    LOCAL CONST Robtarget Tr_meulage_motif_1_369 := [[-197.1254375,6.42979248046875,2.70970288085938],[0.587839766788017,-0.597604018313253,0.388723125784971,-0.382371778977509],[0,0,0,0],[8.999999E+09,8.999999E+09,8.999999E+09,8.999999E+09,8.999999E+09,8.999999E+09]];
    LOCAL CONST Robtarget Tr_meulage_motif_1_370 := [[-197.496625,7.3583505859375,2.7097021484375],[0.587839766788017,-0.597604018313253,0.388723125784971,-0.382371778977509],[0,0,0,0],[8.999999E+09,8.999999E+09,8.999999E+09,8.999999E+09,8.999999E+09,8.999999E+09]];
    LOCAL CONST Robtarget Tr_meulage_motif_1_371 := [[-197.8661875,8.279548828125,2.5990986328125],[0.587839766788017,-0.597604018313253,0.388723125784971,-0.382371778977509],[0,0,0,0],[8.999999E+09,8.999999E+09,8.999999E+09,8.999999E+09,8.999999E+09,8.999999E+09]];
    LOCAL CONST Robtarget Tr_meulage_motif_1_372 := [[-198.2196875,9.1575625,2.38792309570313],[0.587839766788017,-0.597604018313253,0.388723125784971,-0.382371778977509],[0,0,0,0],[8.999999E+09,8.999999E+09,8.999999E+09,8.999999E+09,8.999999E+09,8.999999E+09]];
    LOCAL CONST Robtarget Tr_meulage_motif_1_373 := [[-198.538984375,9.9482470703125,2.11611083984375],[0.587839766788017,-0.597604018313253,0.388723125784971,-0.382371778977509],[0,0,0,0],[8.999999E+09,8.999999E+09,8.999999E+09,8.999999E+09,8.999999E+09,8.999999E+09]];
    LOCAL CONST Robtarget Tr_meulage_motif_1_374 := [[-198.806203125,10.6076689453125,1.81198828125],[0.587839766788017,-0.597604018313253,0.388723125784971,-0.382371778977509],[0,0,0,0],[8.999999E+09,8.999999E+09,8.999999E+09,8.999999E+09,8.999999E+09,8.999999E+09]];
    LOCAL CONST Robtarget Tr_meulage_motif_1_375 := [[-199.196984375,11.5655166015625,1.14949658203125],[0.587839766788017,-0.597604018313253,0.388723125784971,-0.382371778977509],[0,0,0,0],[8.999999E+09,8.999999E+09,8.999999E+09,8.999999E+09,8.999999E+09,8.999999E+09]];
    LOCAL CONST Robtarget Tr_meulage_motif_1_376 := [[-199.541015625,12.3993203125,0.247597717285156],[0.587839766788017,-0.597604018313253,0.388723125784971,-0.382371778977509],[0,0,0,0],[8.999999E+09,8.999999E+09,8.999999E+09,8.999999E+09,8.999999E+09,8.999999E+09]];
    LOCAL CONST Robtarget Tr_meulage_motif_1_377 := [[-199.7503125,12.89178125,-0.798370178222656],[0.587839766788017,-0.597604018313253,0.388723125784971,-0.382371778977509],[0,0,0,0],[8.999999E+09,8.999999E+09,8.999999E+09,8.999999E+09,8.999999E+09,8.999999E+09]];
    LOCAL CONST Robtarget Tr_meulage_motif_1_378 := [[-199.792984375,12.9777431640625,-1.49615588378906],[0.587839766788017,-0.597604018313253,0.388723125784971,-0.382371778977509],[0,0,0,0],[8.999999E+09,8.999999E+09,8.999999E+09,8.999999E+09,8.999999E+09,8.999999E+09]];
    LOCAL CONST Robtarget Tr_meulage_motif_1_379 := [[-199.76965625,12.9004716796875,-2.13255444335937],[0.587839766788017,-0.597604018313253,0.388723125784971,-0.382371778977509],[0,0,0,0],[8.999999E+09,8.999999E+09,8.999999E+09,8.999999E+09,8.999999E+09,8.999999E+09]];
    LOCAL CONST Robtarget Tr_meulage_motif_1_380 := [[-199.738171875,12.8063076171875,-2.64972607421875],[0.587839766788017,-0.597604018313253,0.388723125784971,-0.382371778977509],[0,0,0,0],[8.999999E+09,8.999999E+09,8.999999E+09,8.999999E+09,8.999999E+09,8.999999E+09]];
    LOCAL CONST Robtarget Tr_meulage_motif_1_381 := [[-199.526421875,12.2498720703125,-3.54807690429688],[0.587839766788017,-0.597604018313253,0.388723125784971,-0.382371778977509],[0,0,0,0],[8.999999E+09,8.999999E+09,8.999999E+09,8.999999E+09,8.999999E+09,8.999999E+09]];
    LOCAL CONST Robtarget Tr_meulage_motif_1_382 := [[-199.35234375,11.8015830078125,-3.97934716796875],[0.587839766788017,-0.597604018313253,0.388723125784971,-0.382371778977509],[0,0,0,0],[8.999999E+09,8.999999E+09,8.999999E+09,8.999999E+09,8.999999E+09,8.999999E+09]];
    LOCAL CONST Robtarget Tr_meulage_motif_1_383 := [[-198.956453125,10.7936171875,-4.57071630859375],[0.587839766788017,-0.597604018313253,0.388723125784971,-0.382371778977509],[0,0,0,0],[8.999999E+09,8.999999E+09,8.999999E+09,8.999999E+09,8.999999E+09,8.999999E+09]];
    LOCAL CONST Robtarget Tr_meulage_motif_1_384 := [[-198.65303125,10.025794921875,-4.86619775390625],[0.587839766788017,-0.597604018313253,0.388723125784971,-0.382371778977509],[0,0,0,0],[8.999999E+09,8.999999E+09,8.999999E+09,8.999999E+09,8.999999E+09,8.999999E+09]];
    LOCAL CONST Robtarget Tr_meulage_motif_1_385 := [[-198.309171875,9.1595400390625,-5.0706689453125],[0.587839766788017,-0.597604018313253,0.388723125784971,-0.382371778977509],[0,0,0,0],[8.999999E+09,8.999999E+09,8.999999E+09,8.999999E+09,8.999999E+09,8.999999E+09]];
    LOCAL CONST Robtarget Tr_meulage_motif_1_386 := [[-197.945953125,8.247658203125,-5.17920849609375],[0.587839766788017,-0.597604018313253,0.388723125784971,-0.382371778977509],[0,0,0,0],[8.999999E+09,8.999999E+09,8.999999E+09,8.999999E+09,8.999999E+09,8.999999E+09]];
    LOCAL CONST Robtarget Tr_meulage_motif_1_387 := [[-197.57865625,7.325552734375,-5.28981005859375],[0.587839766788017,-0.597604018313253,0.388723125784971,-0.382371778977509],[0,0,0,0],[8.999999E+09,8.999999E+09,8.999999E+09,8.999999E+09,8.999999E+09,8.999999E+09]];
    LOCAL CONST Robtarget Tr_meulage_motif_1_388 := [[-197.20746875,6.3969951171875,-5.28980908203125],[0.587839766788017,-0.597604018313253,0.388723125784971,-0.382371778977509],[0,0,0,0],[8.999999E+09,8.999999E+09,8.999999E+09,8.999999E+09,8.999999E+09,8.999999E+09]];
    LOCAL CONST Robtarget Tr_meulage_motif_1_389 := [[-196.83628125,5.46843701171875,-5.28980859375],[0.587839766788017,-0.597604018313253,0.388723125784971,-0.382371778977509],[0,0,0,0],[8.999999E+09,8.999999E+09,8.999999E+09,8.999999E+09,8.999999E+09,8.999999E+09]];
    LOCAL CONST Robtarget Tr_meulage_motif_1_390 := [[-196.46509375,4.53987939453125,-5.2898076171875],[0.587839766788017,-0.597604018313253,0.388723125784971,-0.382371778977509],[0,0,0,0],[8.999999E+09,8.999999E+09,8.999999E+09,8.999999E+09,8.999999E+09,8.999999E+09]];
    LOCAL CONST Robtarget Tr_meulage_motif_1_391 := [[-196.09390625,3.61132153320312,-5.289806640625],[0.587839766788017,-0.597604018313253,0.388723125784971,-0.382371778977509],[0,0,0,0],[8.999999E+09,8.999999E+09,8.999999E+09,8.999999E+09,8.999999E+09,8.999999E+09]];
    LOCAL CONST Robtarget Tr_meulage_motif_1_392 := [[-195.72271875,2.682763671875,-5.28980615234375],[0.587839766788017,-0.597604018313253,0.388723125784971,-0.382371778977509],[0,0,0,0],[8.999999E+09,8.999999E+09,8.999999E+09,8.999999E+09,8.999999E+09,8.999999E+09]];
    LOCAL CONST Robtarget Tr_meulage_motif_1_393 := [[-195.35153125,1.75420581054687,-5.28980517578125],[0.587839766788017,-0.597604018313253,0.388723125784971,-0.382371778977509],[0,0,0,0],[8.999999E+09,8.999999E+09,8.999999E+09,8.999999E+09,8.999999E+09,8.999999E+09]];
    LOCAL CONST Robtarget Tr_meulage_motif_1_394 := [[-194.98034375,0.825648010253906,-5.28980419921875],[0.587839766788017,-0.597604018313253,0.388723125784971,-0.382371778977509],[0,0,0,0],[8.999999E+09,8.999999E+09,8.999999E+09,8.999999E+09,8.999999E+09,8.999999E+09]];
    LOCAL CONST Robtarget Tr_meulage_motif_1_395 := [[-194.60915625,-0.102909828186035,-5.2898037109375],[0.587839766788017,-0.597604018313253,0.388723125784971,-0.382371778977509],[0,0,0,0],[8.999999E+09,8.999999E+09,8.999999E+09,8.999999E+09,8.999999E+09,8.999999E+09]];
    LOCAL CONST Robtarget Tr_meulage_motif_1_396 := [[-194.23796875,-1.03146765136719,-5.289802734375],[0.587839766788017,-0.597604018313253,0.388723125784971,-0.382371778977509],[0,0,0,0],[8.999999E+09,8.999999E+09,8.999999E+09,8.999999E+09,8.999999E+09,8.999999E+09]];
    LOCAL CONST Robtarget Tr_meulage_motif_1_397 := [[-193.86678125,-1.96002551269531,-5.2898017578125],[0.587839766788017,-0.597604018313253,0.388723125784971,-0.382371778977509],[0,0,0,0],[8.999999E+09,8.999999E+09,8.999999E+09,8.999999E+09,8.999999E+09,8.999999E+09]];
    LOCAL CONST Robtarget Tr_meulage_motif_1_398 := [[-193.49559375,-2.88858325195313,-5.28980126953125],[0.587839766788017,-0.597604018313253,0.388723125784971,-0.382371778977509],[0,0,0,0],[8.999999E+09,8.999999E+09,8.999999E+09,8.999999E+09,8.999999E+09,8.999999E+09]];
    LOCAL CONST Robtarget Tr_meulage_motif_1_399 := [[-193.12440625,-3.81714111328125,-5.28980029296875],[0.587839766788017,-0.597604018313253,0.388723125784971,-0.382371778977509],[0,0,0,0],[8.999999E+09,8.999999E+09,8.999999E+09,8.999999E+09,8.999999E+09,8.999999E+09]];
    LOCAL CONST Robtarget Tr_meulage_motif_1_400 := [[-192.75321875,-4.74569873046875,-5.28979931640625],[0.587839766788017,-0.597604018313253,0.388723125784971,-0.382371778977509],[0,0,0,0],[8.999999E+09,8.999999E+09,8.999999E+09,8.999999E+09,8.999999E+09,8.999999E+09]];
    LOCAL CONST Robtarget Tr_meulage_motif_1_401 := [[-192.38203125,-5.6742568359375,-5.289798828125],[0.587839766788017,-0.597604018313253,0.388723125784971,-0.382371778977509],[0,0,0,0],[8.999999E+09,8.999999E+09,8.999999E+09,8.999999E+09,8.999999E+09,8.999999E+09]];
    LOCAL CONST Robtarget Tr_meulage_motif_1_402 := [[-192.01084375,-6.602814453125,-5.2897978515625],[0.587839766788017,-0.597604018313253,0.388723125784971,-0.382371778977509],[0,0,0,0],[8.999999E+09,8.999999E+09,8.999999E+09,8.999999E+09,8.999999E+09,8.999999E+09]];
    LOCAL CONST Robtarget Tr_meulage_motif_1_403 := [[-191.63965625,-7.53137255859375,-5.289796875],[0.587839766788017,-0.597604018313253,0.388723125784971,-0.382371778977509],[0,0,0,0],[8.999999E+09,8.999999E+09,8.999999E+09,8.999999E+09,8.999999E+09,8.999999E+09]];
    LOCAL CONST Robtarget Tr_meulage_motif_1_404 := [[-191.268453125,-8.4599306640625,-5.28979638671875],[0.587839766788017,-0.597604018313253,0.388723125784971,-0.382371778977509],[0,0,0,0],[8.999999E+09,8.999999E+09,8.999999E+09,8.999999E+09,8.999999E+09,8.999999E+09]];
    LOCAL CONST Robtarget Tr_meulage_motif_1_405 := [[-190.897265625,-9.38848828125,-5.28979541015625],[0.587839766788017,-0.597604018313253,0.388723125784971,-0.382371778977509],[0,0,0,0],[8.999999E+09,8.999999E+09,8.999999E+09,8.999999E+09,8.999999E+09,8.999999E+09]];
    LOCAL CONST Robtarget Tr_meulage_motif_1_406 := [[-190.526078125,-10.3170458984375,-5.28979443359375],[0.587839766788017,-0.597604018313253,0.388723125784971,-0.382371778977509],[0,0,0,0],[8.999999E+09,8.999999E+09,8.999999E+09,8.999999E+09,8.999999E+09,8.999999E+09]];
    LOCAL CONST Robtarget Tr_meulage_motif_1_407 := [[-190.154890625,-11.245603515625,-5.28979345703125],[0.587839766788017,-0.597604018313253,0.388723125784971,-0.382371778977509],[0,0,0,0],[8.999999E+09,8.999999E+09,8.999999E+09,8.999999E+09,8.999999E+09,8.999999E+09]];
    LOCAL CONST Robtarget Tr_meulage_motif_1_408 := [[-189.783703125,-12.1741611328125,-5.28979296875],[0.587839766788017,-0.597604018313253,0.388723125784971,-0.382371778977509],[0,0,0,0],[8.999999E+09,8.999999E+09,8.999999E+09,8.999999E+09,8.999999E+09,8.999999E+09]];
    LOCAL CONST Robtarget Tr_meulage_motif_1_409 := [[-189.412515625,-13.1027197265625,-5.2897919921875],[0.587839766788017,-0.597604018313253,0.388723125784971,-0.382371778977509],[0,0,0,0],[8.999999E+09,8.999999E+09,8.999999E+09,8.999999E+09,8.999999E+09,8.999999E+09]];
    LOCAL CONST Robtarget Tr_meulage_motif_1_410 := [[-189.041328125,-14.03127734375,-5.289791015625],[0.587839766788017,-0.597604018313253,0.388723125784971,-0.382371778977509],[0,0,0,0],[8.999999E+09,8.999999E+09,8.999999E+09,8.999999E+09,8.999999E+09,8.999999E+09]];
    LOCAL CONST Robtarget Tr_meulage_motif_1_411 := [[-188.670140625,-14.9598349609375,-5.28979052734375],[0.587839766788017,-0.597604018313253,0.388723125784971,-0.382371778977509],[0,0,0,0],[8.999999E+09,8.999999E+09,8.999999E+09,8.999999E+09,8.999999E+09,8.999999E+09]];
    LOCAL CONST Robtarget Tr_meulage_motif_1_412 := [[-188.298953125,-15.888392578125,-5.28978955078125],[0.587839766788017,-0.597604018313253,0.388723125784971,-0.382371778977509],[0,0,0,0],[8.999999E+09,8.999999E+09,8.999999E+09,8.999999E+09,8.999999E+09,8.999999E+09]];
    LOCAL CONST Robtarget Tr_meulage_motif_1_413 := [[-187.927765625,-16.816951171875,-5.28978857421875],[0.587839766788017,-0.597604018313253,0.388723125784971,-0.382371778977509],[0,0,0,0],[8.999999E+09,8.999999E+09,8.999999E+09,8.999999E+09,8.999999E+09,8.999999E+09]];
    LOCAL CONST Robtarget Tr_meulage_motif_1_414 := [[-187.556578125,-17.7455078125,-5.2897880859375],[0.587839766788017,-0.597604018313253,0.388723125784971,-0.382371778977509],[0,0,0,0],[8.999999E+09,8.999999E+09,8.999999E+09,8.999999E+09,8.999999E+09,8.999999E+09]];
    LOCAL CONST Robtarget Tr_meulage_motif_1_415 := [[-187.185390625,-18.67406640625,-5.289787109375],[0.587839766788017,-0.597604018313253,0.388723125784971,-0.382371778977509],[0,0,0,0],[8.999999E+09,8.999999E+09,8.999999E+09,8.999999E+09,8.999999E+09,8.999999E+09]];
    LOCAL CONST Robtarget Tr_meulage_motif_1_416 := [[-186.814203125,-19.602625,-5.2897861328125],[0.587839766788017,-0.597604018313253,0.388723125784971,-0.382371778977509],[0,0,0,0],[8.999999E+09,8.999999E+09,8.999999E+09,8.999999E+09,8.999999E+09,8.999999E+09]];
    LOCAL CONST Robtarget Tr_meulage_motif_1_417 := [[-186.443015625,-20.531181640625,-5.28978564453125],[0.587839766788017,-0.597604018313253,0.388723125784971,-0.382371778977509],[0,0,0,0],[8.999999E+09,8.999999E+09,8.999999E+09,8.999999E+09,8.999999E+09,8.999999E+09]];
    LOCAL CONST Robtarget Tr_meulage_motif_1_418 := [[-186.071828125,-21.459740234375,-5.28978466796875],[0.587839766788017,-0.597604018313253,0.388723125784971,-0.382371778977509],[0,0,0,0],[8.999999E+09,8.999999E+09,8.999999E+09,8.999999E+09,8.999999E+09,8.999999E+09]];
    LOCAL CONST Robtarget Tr_meulage_motif_1_419 := [[-185.700640625,-22.388296875,-5.28978369140625],[0.587839766788017,-0.597604018313253,0.388723125784971,-0.382371778977509],[0,0,0,0],[8.999999E+09,8.999999E+09,8.999999E+09,8.999999E+09,8.999999E+09,8.999999E+09]];
    LOCAL CONST Robtarget Tr_meulage_motif_1_420 := [[-185.329453125,-23.31685546875,-5.289783203125],[0.587839766788017,-0.597604018313253,0.388723125784971,-0.382371778977509],[0,0,0,0],[8.999999E+09,8.999999E+09,8.999999E+09,8.999999E+09,8.999999E+09,8.999999E+09]];
    LOCAL CONST Robtarget Tr_meulage_motif_1_421 := [[-184.958265625,-24.2454140625,-5.2897822265625],[0.587839766788017,-0.597604018313253,0.388723125784971,-0.382371778977509],[0,0,0,0],[8.999999E+09,8.999999E+09,8.999999E+09,8.999999E+09,8.999999E+09,8.999999E+09]];
    LOCAL CONST Robtarget Tr_meulage_motif_1_422 := [[-184.587078125,-25.173970703125,-5.28978125],[0.587839766788017,-0.597604018313253,0.388723125784971,-0.382371778977509],[0,0,0,0],[8.999999E+09,8.999999E+09,8.999999E+09,8.999999E+09,8.999999E+09,8.999999E+09]];
    LOCAL CONST Robtarget Tr_meulage_motif_1_423 := [[-184.215890625,-26.102529296875,-5.28978076171875],[0.587839766788017,-0.597604018313253,0.388723125784971,-0.382371778977509],[0,0,0,0],[8.999999E+09,8.999999E+09,8.999999E+09,8.999999E+09,8.999999E+09,8.999999E+09]];
    LOCAL CONST Robtarget Tr_meulage_motif_1_424 := [[-183.844703125,-27.0310859375,-5.28977978515625],[0.587839766788017,-0.597604018313253,0.388723125784971,-0.382371778977509],[0,0,0,0],[8.999999E+09,8.999999E+09,8.999999E+09,8.999999E+09,8.999999E+09,8.999999E+09]];
    LOCAL CONST Robtarget Tr_meulage_motif_1_425 := [[-183.473515625,-27.95964453125,-5.28977880859375],[0.587839766788017,-0.597604018313253,0.388723125784971,-0.382371778977509],[0,0,0,0],[8.999999E+09,8.999999E+09,8.999999E+09,8.999999E+09,8.999999E+09,8.999999E+09]];
    LOCAL CONST Robtarget Tr_meulage_motif_1_426 := [[-183.102328125,-28.888203125,-5.28977783203125],[0.587839766788017,-0.597604018313253,0.388723125784971,-0.382371778977509],[0,0,0,0],[8.999999E+09,8.999999E+09,8.999999E+09,8.999999E+09,8.999999E+09,8.999999E+09]];
    LOCAL CONST Robtarget Tr_meulage_motif_1_427 := [[-182.731140625,-29.816759765625,-5.28977734375],[0.587839766788017,-0.597604018313253,0.388723125784971,-0.382371778977509],[0,0,0,0],[8.999999E+09,8.999999E+09,8.999999E+09,8.999999E+09,8.999999E+09,8.999999E+09]];
    LOCAL CONST Robtarget Tr_meulage_motif_1_428 := [[-182.359953125,-30.745318359375,-5.2897763671875],[0.587839766788017,-0.597604018313253,0.388723125784971,-0.382371778977509],[0,0,0,0],[8.999999E+09,8.999999E+09,8.999999E+09,8.999999E+09,8.999999E+09,8.999999E+09]];
    LOCAL CONST Robtarget Tr_meulage_motif_1_429 := [[-181.988765625,-31.673875,-5.289775390625],[0.587839766788017,-0.597604018313253,0.388723125784971,-0.382371778977509],[0,0,0,0],[8.999999E+09,8.999999E+09,8.999999E+09,8.999999E+09,8.999999E+09,8.999999E+09]];
    LOCAL CONST Robtarget Tr_meulage_motif_1_430 := [[-181.617578125,-32.60243359375,-5.28977490234375],[0.587839766788017,-0.597604018313253,0.388723125784971,-0.382371778977509],[0,0,0,0],[8.999999E+09,8.999999E+09,8.999999E+09,8.999999E+09,8.999999E+09,8.999999E+09]];
    LOCAL CONST Robtarget Tr_meulage_motif_1_431 := [[-181.246390625,-33.5309921875,-5.28977392578125],[0.587839766788017,-0.597604018313253,0.388723125784971,-0.382371778977509],[0,0,0,0],[8.999999E+09,8.999999E+09,8.999999E+09,8.999999E+09,8.999999E+09,8.999999E+09]];
    LOCAL CONST Robtarget Tr_meulage_motif_1_432 := [[-180.875203125,-34.45955078125,-5.28977294921875],[0.587839766788017,-0.597604018313253,0.388723125784971,-0.382371778977509],[0,0,0,0],[8.999999E+09,8.999999E+09,8.999999E+09,8.999999E+09,8.999999E+09,8.999999E+09]];
    LOCAL CONST Robtarget Tr_meulage_motif_1_433 := [[-180.504015625,-35.38810546875,-5.2897724609375],[0.587839766788017,-0.597604018313253,0.388723125784971,-0.382371778977509],[0,0,0,0],[8.999999E+09,8.999999E+09,8.999999E+09,8.999999E+09,8.999999E+09,8.999999E+09]];
    LOCAL CONST Robtarget Tr_meulage_motif_1_434 := [[-180.132828125,-36.3166640625,-5.289771484375],[0.587839766788017,-0.597604018313253,0.388723125784971,-0.382371778977509],[0,0,0,0],[8.999999E+09,8.999999E+09,8.999999E+09,8.999999E+09,8.999999E+09,8.999999E+09]];
    LOCAL CONST Robtarget Tr_meulage_motif_1_435 := [[-179.761640625,-37.24522265625,-5.2897705078125],[0.587839766788017,-0.597604018313253,0.388723125784971,-0.382371778977509],[0,0,0,0],[8.999999E+09,8.999999E+09,8.999999E+09,8.999999E+09,8.999999E+09,8.999999E+09]];
    LOCAL CONST Robtarget Tr_meulage_motif_1_436 := [[-179.390453125,-38.17378125,-5.28977001953125],[0.587839766788017,-0.597604018313253,0.388723125784971,-0.382371778977509],[0,0,0,0],[8.999999E+09,8.999999E+09,8.999999E+09,8.999999E+09,8.999999E+09,8.999999E+09]];
    LOCAL CONST Robtarget Tr_meulage_motif_1_437 := [[-179.02315625,-39.09588671875,-5.40037158203125],[0.587839766788017,-0.597604018313253,0.388723125784971,-0.382371778977509],[0,0,0,0],[8.999999E+09,8.999999E+09,8.999999E+09,8.999999E+09,8.999999E+09,8.999999E+09]];
    LOCAL CONST Robtarget Tr_meulage_motif_1_438 := [[-178.659921875,-40.00776953125,-5.5089111328125],[0.587839766788017,-0.597604018313253,0.388723125784971,-0.382371778977509],[0,0,0,0],[8.999999E+09,8.999999E+09,8.999999E+09,8.999999E+09,8.999999E+09,8.999999E+09]];
    LOCAL CONST Robtarget Tr_meulage_motif_1_439 := [[-178.297125,-40.9182109375,-5.605623046875],[0.587839766788017,-0.597604018313253,0.388723125784971,-0.382371778977509],[0,0,0,0],[8.999999E+09,8.999999E+09,8.999999E+09,8.999999E+09,8.999999E+09,8.999999E+09]];
    LOCAL CONST Robtarget Tr_meulage_motif_1_440 := [[-177.940921875,-41.81337890625,-5.74241064453125],[0.587839766788017,-0.597604018313253,0.388723125784971,-0.382371778977509],[0,0,0,0],[8.999999E+09,8.999999E+09,8.999999E+09,8.999999E+09,8.999999E+09,8.999999E+09]];
    LOCAL CONST Robtarget Tr_meulage_motif_1_441 := [[-177.515703125,-42.88446875,-5.99027001953125],[0.587839766788017,-0.597604018313253,0.388723125784971,-0.382371778977509],[0,0,0,0],[8.999999E+09,8.999999E+09,8.999999E+09,8.999999E+09,8.999999E+09,8.999999E+09]];
    LOCAL CONST Robtarget Tr_meulage_motif_1_442 := [[-177.1755,-43.74487890625,-6.305171875],[0.587839766788017,-0.597604018313253,0.388723125784971,-0.382371778977509],[0,0,0,0],[8.999999E+09,8.999999E+09,8.999999E+09,8.999999E+09,8.999999E+09,8.999999E+09]];

    !Tr_meulage_motif_2 : Meulage d'un motif
    LOCAL CONST Robtarget Tr_meulage_motif_2_0 := [[111.493109375,113.3949609375,1.99855541992188],[-0.000489514218315733,0.0476030487198184,-0.010271051450657,-0.998813403809994],[0,0,0,0],[8.999999E+09,8.999999E+09,8.999999E+09,8.999999E+09,8.999999E+09,8.999999E+09]];
    LOCAL CONST Robtarget Tr_meulage_motif_2_1 := [[110.787296875,112.68659375,1.99164038085938],[-0.000489514218315733,0.0476030487198184,-0.010271051450657,-0.998813403809994],[0,0,0,0],[8.999999E+09,8.999999E+09,8.999999E+09,8.999999E+09,8.999999E+09,8.999999E+09]];
    LOCAL CONST Robtarget Tr_meulage_motif_2_2 := [[110.081484375,111.978234375,1.98472546386719],[-0.000489514218315733,0.0476030487198184,-0.010271051450657,-0.998813403809994],[0,0,0,0],[8.999999E+09,8.999999E+09,8.999999E+09,8.999999E+09,8.999999E+09,8.999999E+09]];
    LOCAL CONST Robtarget Tr_meulage_motif_2_3 := [[109.3756640625,111.2698671875,1.977810546875],[-0.000489514218315733,0.0476030487198184,-0.010271051450657,-0.998813403809994],[0,0,0,0],[8.999999E+09,8.999999E+09,8.999999E+09,8.999999E+09,8.999999E+09,8.999999E+09]];
    LOCAL CONST Robtarget Tr_meulage_motif_2_4 := [[108.6698515625,110.5615078125,1.9708955078125],[-0.000489514218315733,0.0476030487198184,-0.010271051450657,-0.998813403809994],[0,0,0,0],[8.999999E+09,8.999999E+09,8.999999E+09,8.999999E+09,8.999999E+09,8.999999E+09]];
    LOCAL CONST Robtarget Tr_meulage_motif_2_5 := [[107.9640390625,109.8531484375,1.96398059082031],[-0.000489514218315733,0.0476030487198184,-0.010271051450657,-0.998813403809994],[0,0,0,0],[8.999999E+09,8.999999E+09,8.999999E+09,8.999999E+09,8.999999E+09,8.999999E+09]];
    LOCAL CONST Robtarget Tr_meulage_motif_2_6 := [[107.25821875,109.14478125,1.95706567382813],[-0.000489514218315733,0.0476030487198184,-0.010271051450657,-0.998813403809994],[0,0,0,0],[8.999999E+09,8.999999E+09,8.999999E+09,8.999999E+09,8.999999E+09,8.999999E+09]];
    LOCAL CONST Robtarget Tr_meulage_motif_2_7 := [[106.55240625,108.436421875,1.95015075683594],[-0.000489514218315733,0.0476030487198184,-0.010271051450657,-0.998813403809994],[0,0,0,0],[8.999999E+09,8.999999E+09,8.999999E+09,8.999999E+09,8.999999E+09,8.999999E+09]];
    LOCAL CONST Robtarget Tr_meulage_motif_2_8 := [[105.84659375,107.7280546875,1.94323571777344],[-0.000489514218315733,0.0476030487198184,-0.010271051450657,-0.998813403809994],[0,0,0,0],[8.999999E+09,8.999999E+09,8.999999E+09,8.999999E+09,8.999999E+09,8.999999E+09]];
    LOCAL CONST Robtarget Tr_meulage_motif_2_9 := [[105.1407734375,107.0196953125,1.93632080078125],[-0.000489514218315733,0.0476030487198184,-0.010271051450657,-0.998813403809994],[0,0,0,0],[8.999999E+09,8.999999E+09,8.999999E+09,8.999999E+09,8.999999E+09,8.999999E+09]];
    LOCAL CONST Robtarget Tr_meulage_motif_2_10 := [[104.4349609375,106.3113359375,1.92940588378906],[-0.000489514218315733,0.0476030487198184,-0.010271051450657,-0.998813403809994],[0,0,0,0],[8.999999E+09,8.999999E+09,8.999999E+09,8.999999E+09,8.999999E+09,8.999999E+09]];
    LOCAL CONST Robtarget Tr_meulage_motif_2_11 := [[103.7291484375,105.60296875,1.92249084472656],[-0.000489514218315733,0.0476030487198184,-0.010271051450657,-0.998813403809994],[0,0,0,0],[8.999999E+09,8.999999E+09,8.999999E+09,8.999999E+09,8.999999E+09,8.999999E+09]];
    LOCAL CONST Robtarget Tr_meulage_motif_2_12 := [[103.023328125,104.894609375,1.91557592773438],[-0.000489514218315733,0.0476030487198184,-0.010271051450657,-0.998813403809994],[0,0,0,0],[8.999999E+09,8.999999E+09,8.999999E+09,8.999999E+09,8.999999E+09,8.999999E+09]];
    LOCAL CONST Robtarget Tr_meulage_motif_2_13 := [[102.317515625,104.1862421875,1.90866101074219],[-0.000489514218315733,0.0476030487198184,-0.010271051450657,-0.998813403809994],[0,0,0,0],[8.999999E+09,8.999999E+09,8.999999E+09,8.999999E+09,8.999999E+09,8.999999E+09]];
    LOCAL CONST Robtarget Tr_meulage_motif_2_14 := [[101.611703125,103.4778828125,1.90174597167969],[-0.000489514218315733,0.0476030487198184,-0.010271051450657,-0.998813403809994],[0,0,0,0],[8.999999E+09,8.999999E+09,8.999999E+09,8.999999E+09,8.999999E+09,8.999999E+09]];
    LOCAL CONST Robtarget Tr_meulage_motif_2_15 := [[100.9058828125,102.7695234375,1.8948310546875],[-0.000489514218315733,0.0476030487198184,-0.010271051450657,-0.998813403809994],[0,0,0,0],[8.999999E+09,8.999999E+09,8.999999E+09,8.999999E+09,8.999999E+09,8.999999E+09]];
    LOCAL CONST Robtarget Tr_meulage_motif_2_16 := [[100.2000703125,102.06115625,1.88791613769531],[-0.000489514218315733,0.0476030487198184,-0.010271051450657,-0.998813403809994],[0,0,0,0],[8.999999E+09,8.999999E+09,8.999999E+09,8.999999E+09,8.999999E+09,8.999999E+09]];
    LOCAL CONST Robtarget Tr_meulage_motif_2_17 := [[99.4942578125,101.352796875,1.88100122070313],[-0.000489514218315733,0.0476030487198184,-0.010271051450657,-0.998813403809994],[0,0,0,0],[8.999999E+09,8.999999E+09,8.999999E+09,8.999999E+09,8.999999E+09,8.999999E+09]];
    LOCAL CONST Robtarget Tr_meulage_motif_2_18 := [[98.7884375,100.6444375,1.87408618164063],[-0.000489514218315733,0.0476030487198184,-0.010271051450657,-0.998813403809994],[0,0,0,0],[8.999999E+09,8.999999E+09,8.999999E+09,8.999999E+09,8.999999E+09,8.999999E+09]];
    LOCAL CONST Robtarget Tr_meulage_motif_2_19 := [[98.082625,99.9360703125,1.86717126464844],[-0.000489514218315733,0.0476030487198184,-0.010271051450657,-0.998813403809994],[0,0,0,0],[8.999999E+09,8.999999E+09,8.999999E+09,8.999999E+09,8.999999E+09,8.999999E+09]];
    LOCAL CONST Robtarget Tr_meulage_motif_2_20 := [[97.3768125,99.2277109375,1.86025634765625],[-0.000489514218315733,0.0476030487198184,-0.010271051450657,-0.998813403809994],[0,0,0,0],[8.999999E+09,8.999999E+09,8.999999E+09,8.999999E+09,8.999999E+09,8.999999E+09]];
    LOCAL CONST Robtarget Tr_meulage_motif_2_21 := [[96.671,98.51934375,1.85334130859375],[-0.000489514218315733,0.0476030487198184,-0.010271051450657,-0.998813403809994],[0,0,0,0],[8.999999E+09,8.999999E+09,8.999999E+09,8.999999E+09,8.999999E+09,8.999999E+09]];
    LOCAL CONST Robtarget Tr_meulage_motif_2_22 := [[95.9651796875,97.810984375,1.84642639160156],[-0.000489514218315733,0.0476030487198184,-0.010271051450657,-0.998813403809994],[0,0,0,0],[8.999999E+09,8.999999E+09,8.999999E+09,8.999999E+09,8.999999E+09,8.999999E+09]];
    LOCAL CONST Robtarget Tr_meulage_motif_2_23 := [[95.2593671875,97.102625,1.83951147460938],[-0.000489514218315733,0.0476030487198184,-0.010271051450657,-0.998813403809994],[0,0,0,0],[8.999999E+09,8.999999E+09,8.999999E+09,8.999999E+09,8.999999E+09,8.999999E+09]];
    LOCAL CONST Robtarget Tr_meulage_motif_2_24 := [[94.5535546875,96.3942578125,1.83259655761719],[-0.000489514218315733,0.0476030487198184,-0.010271051450657,-0.998813403809994],[0,0,0,0],[8.999999E+09,8.999999E+09,8.999999E+09,8.999999E+09,8.999999E+09,8.999999E+09]];
    LOCAL CONST Robtarget Tr_meulage_motif_2_25 := [[93.847734375,95.6858984375,1.82568151855469],[-0.000489514218315733,0.0476030487198184,-0.010271051450657,-0.998813403809994],[0,0,0,0],[8.999999E+09,8.999999E+09,8.999999E+09,8.999999E+09,8.999999E+09,8.999999E+09]];
    LOCAL CONST Robtarget Tr_meulage_motif_2_26 := [[93.141921875,94.97753125,1.8187666015625],[-0.000489514218315733,0.0476030487198184,-0.010271051450657,-0.998813403809994],[0,0,0,0],[8.999999E+09,8.999999E+09,8.999999E+09,8.999999E+09,8.999999E+09,8.999999E+09]];
    LOCAL CONST Robtarget Tr_meulage_motif_2_27 := [[92.436109375,94.269171875,1.81185168457031],[-0.000489514218315733,0.0476030487198184,-0.010271051450657,-0.998813403809994],[0,0,0,0],[8.999999E+09,8.999999E+09,8.999999E+09,8.999999E+09,8.999999E+09,8.999999E+09]];
    LOCAL CONST Robtarget Tr_meulage_motif_2_28 := [[91.7302890625,93.5608125,1.80493664550781],[-0.000489514218315733,0.0476030487198184,-0.010271051450657,-0.998813403809994],[0,0,0,0],[8.999999E+09,8.999999E+09,8.999999E+09,8.999999E+09,8.999999E+09,8.999999E+09]];
    LOCAL CONST Robtarget Tr_meulage_motif_2_29 := [[91.0244765625,92.8524453125,1.79802172851563],[-0.000489514218315733,0.0476030487198184,-0.010271051450657,-0.998813403809994],[0,0,0,0],[8.999999E+09,8.999999E+09,8.999999E+09,8.999999E+09,8.999999E+09,8.999999E+09]];
    LOCAL CONST Robtarget Tr_meulage_motif_2_30 := [[90.3186640625,92.1440859375,1.79110681152344],[-0.000489514218315733,0.0476030487198184,-0.010271051450657,-0.998813403809994],[0,0,0,0],[8.999999E+09,8.999999E+09,8.999999E+09,8.999999E+09,8.999999E+09,8.999999E+09]];
    LOCAL CONST Robtarget Tr_meulage_motif_2_31 := [[89.61284375,91.43571875,1.78419177246094],[-0.000489514218315733,0.0476030487198184,-0.010271051450657,-0.998813403809994],[0,0,0,0],[8.999999E+09,8.999999E+09,8.999999E+09,8.999999E+09,8.999999E+09,8.999999E+09]];
    LOCAL CONST Robtarget Tr_meulage_motif_2_32 := [[88.90703125,90.727359375,1.77727685546875],[-0.000489514218315733,0.0476030487198184,-0.010271051450657,-0.998813403809994],[0,0,0,0],[8.999999E+09,8.999999E+09,8.999999E+09,8.999999E+09,8.999999E+09,8.999999E+09]];
    LOCAL CONST Robtarget Tr_meulage_motif_2_33 := [[88.20121875,90.019,1.77036193847656],[-0.000489514218315733,0.0476030487198184,-0.010271051450657,-0.998813403809994],[0,0,0,0],[8.999999E+09,8.999999E+09,8.999999E+09,8.999999E+09,8.999999E+09,8.999999E+09]];
    LOCAL CONST Robtarget Tr_meulage_motif_2_34 := [[87.4953984375,89.3106328125,1.76344702148437],[-0.000489514218315733,0.0476030487198184,-0.010271051450657,-0.998813403809994],[0,0,0,0],[8.999999E+09,8.999999E+09,8.999999E+09,8.999999E+09,8.999999E+09,8.999999E+09]];
    LOCAL CONST Robtarget Tr_meulage_motif_2_35 := [[86.7895859375,88.6022734375,1.75653198242188],[-0.000489514218315733,0.0476030487198184,-0.010271051450657,-0.998813403809994],[0,0,0,0],[8.999999E+09,8.999999E+09,8.999999E+09,8.999999E+09,8.999999E+09,8.999999E+09]];
    LOCAL CONST Robtarget Tr_meulage_motif_2_36 := [[86.0837734375,87.89390625,1.74961706542969],[-0.000489514218315733,0.0476030487198184,-0.010271051450657,-0.998813403809994],[0,0,0,0],[8.999999E+09,8.999999E+09,8.999999E+09,8.999999E+09,8.999999E+09,8.999999E+09]];
    LOCAL CONST Robtarget Tr_meulage_motif_2_37 := [[85.377953125,87.185546875,1.7427021484375],[-0.000489514218315733,0.0476030487198184,-0.010271051450657,-0.998813403809994],[0,0,0,0],[8.999999E+09,8.999999E+09,8.999999E+09,8.999999E+09,8.999999E+09,8.999999E+09]];
    LOCAL CONST Robtarget Tr_meulage_motif_2_38 := [[84.672140625,86.4771875,1.735787109375],[-0.000489514218315733,0.0476030487198184,-0.010271051450657,-0.998813403809994],[0,0,0,0],[8.999999E+09,8.999999E+09,8.999999E+09,8.999999E+09,8.999999E+09,8.999999E+09]];
    LOCAL CONST Robtarget Tr_meulage_motif_2_39 := [[84.049921875,85.6960390625,1.72813989257813],[-0.000489514218315733,0.0476030487198184,-0.010271051450657,-0.998813403809994],[0,0,0,0],[8.999999E+09,8.999999E+09,8.999999E+09,8.999999E+09,8.999999E+09,8.999999E+09]];
    LOCAL CONST Robtarget Tr_meulage_motif_2_40 := [[83.53146875,84.876515625,1.72009826660156],[-0.000489514218315733,0.0476030487198184,-0.010271051450657,-0.998813403809994],[0,0,0,0],[8.999999E+09,8.999999E+09,8.999999E+09,8.999999E+09,8.999999E+09,8.999999E+09]];
    LOCAL CONST Robtarget Tr_meulage_motif_2_41 := [[83.1221796875,84.080625,1.712275390625],[-0.000489514218315733,0.0476030487198184,-0.010271051450657,-0.998813403809994],[0,0,0,0],[8.999999E+09,8.999999E+09,8.999999E+09,8.999999E+09,8.999999E+09,8.999999E+09]];
    LOCAL CONST Robtarget Tr_meulage_motif_2_42 := [[82.7883359375,83.354640625,1.70513415527344],[-0.000489514218315733,0.0476030487198184,-0.010271051450657,-0.998813403809994],[0,0,0,0],[8.999999E+09,8.999999E+09,8.999999E+09,8.999999E+09,8.999999E+09,8.999999E+09]];
    LOCAL CONST Robtarget Tr_meulage_motif_2_43 := [[82.44765625,82.13984375,1.69315417480469],[-0.000489514218315733,0.0476030487198184,-0.010271051450657,-0.998813403809994],[0,0,0,0],[8.999999E+09,8.999999E+09,8.999999E+09,8.999999E+09,8.999999E+09,8.999999E+09]];
    LOCAL CONST Robtarget Tr_meulage_motif_2_44 := [[82.3254609375,80.8163125,1.68006726074219],[-0.000489514218315733,0.0476030487198184,-0.010271051450657,-0.998813403809994],[0,0,0,0],[8.999999E+09,8.999999E+09,8.999999E+09,8.999999E+09,8.999999E+09,8.999999E+09]];
    LOCAL CONST Robtarget Tr_meulage_motif_2_45 := [[82.452484375,79.493234375,1.66694995117188],[-0.000489514218315733,0.0476030487198184,-0.010271051450657,-0.998813403809994],[0,0,0,0],[8.999999E+09,8.999999E+09,8.999999E+09,8.999999E+09,8.999999E+09,8.999999E+09]];
    LOCAL CONST Robtarget Tr_meulage_motif_2_46 := [[82.898640625,78.35965625,1.65566455078125],[-0.000489514218315733,0.0476030487198184,-0.010271051450657,-0.998813403809994],[0,0,0,0],[8.999999E+09,8.999999E+09,8.999999E+09,8.999999E+09,8.999999E+09,8.999999E+09]];
    LOCAL CONST Robtarget Tr_meulage_motif_2_47 := [[83.3725625,77.8492890625,1.65054541015625],[-0.000489514218315733,0.0476030487198184,-0.010271051450657,-0.998813403809994],[0,0,0,0],[8.999999E+09,8.999999E+09,8.999999E+09,8.999999E+09,8.999999E+09,8.999999E+09]];
    LOCAL CONST Robtarget Tr_meulage_motif_2_48 := [[83.840984375,77.38259375,1.64585949707031],[-0.000489514218315733,0.0476030487198184,-0.010271051450657,-0.998813403809994],[0,0,0,0],[8.999999E+09,8.999999E+09,8.999999E+09,8.999999E+09,8.999999E+09,8.999999E+09]];
    LOCAL CONST Robtarget Tr_meulage_motif_2_49 := [[84.34803125,76.954875,1.64155407714844],[-0.000489514218315733,0.0476030487198184,-0.010271051450657,-0.998813403809994],[0,0,0,0],[8.999999E+09,8.999999E+09,8.999999E+09,8.999999E+09,8.999999E+09,8.999999E+09]];
    LOCAL CONST Robtarget Tr_meulage_motif_2_50 := [[85.48015625,76.530203125,1.63719165039062],[-0.000489514218315733,0.0476030487198184,-0.010271051450657,-0.998813403809994],[0,0,0,0],[8.999999E+09,8.999999E+09,8.999999E+09,8.999999E+09,8.999999E+09,8.999999E+09]];
    LOCAL CONST Robtarget Tr_meulage_motif_2_51 := [[86.7978671875,76.426546875,1.63598168945312],[-0.000489514218315733,0.0476030487198184,-0.010271051450657,-0.998813403809994],[0,0,0,0],[8.999999E+09,8.999999E+09,8.999999E+09,8.999999E+09,8.999999E+09,8.999999E+09]];
    LOCAL CONST Robtarget Tr_meulage_motif_2_52 := [[88.107375,76.5664921875,1.63718469238281],[-0.000489514218315733,0.0476030487198184,-0.010271051450657,-0.998813403809994],[0,0,0,0],[8.999999E+09,8.999999E+09,8.999999E+09,8.999999E+09,8.999999E+09,8.999999E+09]];
    LOCAL CONST Robtarget Tr_meulage_motif_2_53 := [[88.8726875,76.773890625,1.63913146972656],[-0.000489514218315733,0.0476030487198184,-0.010271051450657,-0.998813403809994],[0,0,0,0],[8.999999E+09,8.999999E+09,8.999999E+09,8.999999E+09,8.999999E+09,8.999999E+09]];
    LOCAL CONST Robtarget Tr_meulage_motif_2_54 := [[90.0354921875,77.2501953125,1.64368505859375],[-0.000489514218315733,0.0476030487198184,-0.010271051450657,-0.998813403809994],[0,0,0,0],[8.999999E+09,8.999999E+09,8.999999E+09,8.999999E+09,8.999999E+09,8.999999E+09]];
    LOCAL CONST Robtarget Tr_meulage_motif_2_55 := [[90.819015625,77.662390625,1.64765698242187],[-0.000489514218315733,0.0476030487198184,-0.010271051450657,-0.998813403809994],[0,0,0,0],[8.999999E+09,8.999999E+09,8.999999E+09,8.999999E+09,8.999999E+09,8.999999E+09]];
    LOCAL CONST Robtarget Tr_meulage_motif_2_56 := [[91.6216796875,78.1782734375,1.65265270996094],[-0.000489514218315733,0.0476030487198184,-0.010271051450657,-0.998813403809994],[0,0,0,0],[8.999999E+09,8.999999E+09,8.999999E+09,8.999999E+09,8.999999E+09,8.999999E+09]];
    LOCAL CONST Robtarget Tr_meulage_motif_2_57 := [[92.39140625,78.7969375,1.65867065429687],[-0.000489514218315733,0.0476030487198184,-0.010271051450657,-0.998813403809994],[0,0,0,0],[8.999999E+09,8.999999E+09,8.999999E+09,8.999999E+09,8.999999E+09,8.999999E+09]];
    LOCAL CONST Robtarget Tr_meulage_motif_2_58 := [[93.1703125,79.4219765625,1.66475048828125],[-0.000489514218315733,0.0476030487198184,-0.010271051450657,-0.998813403809994],[0,0,0,0],[8.999999E+09,8.999999E+09,8.999999E+09,8.999999E+09,8.999999E+09,8.999999E+09]];
    LOCAL CONST Robtarget Tr_meulage_motif_2_59 := [[93.8761328125,80.1303359375,1.67166540527344],[-0.000489514218315733,0.0476030487198184,-0.010271051450657,-0.998813403809994],[0,0,0,0],[8.999999E+09,8.999999E+09,8.999999E+09,8.999999E+09,8.999999E+09,8.999999E+09]];
    LOCAL CONST Robtarget Tr_meulage_motif_2_60 := [[94.5819453125,80.8386953125,1.67858032226563],[-0.000489514218315733,0.0476030487198184,-0.010271051450657,-0.998813403809994],[0,0,0,0],[8.999999E+09,8.999999E+09,8.999999E+09,8.999999E+09,8.999999E+09,8.999999E+09]];
    LOCAL CONST Robtarget Tr_meulage_motif_2_61 := [[95.2877578125,81.5470625,1.68549523925781],[-0.000489514218315733,0.0476030487198184,-0.010271051450657,-0.998813403809994],[0,0,0,0],[8.999999E+09,8.999999E+09,8.999999E+09,8.999999E+09,8.999999E+09,8.999999E+09]];
    LOCAL CONST Robtarget Tr_meulage_motif_2_62 := [[95.993578125,82.255421875,1.69241027832031],[-0.000489514218315733,0.0476030487198184,-0.010271051450657,-0.998813403809994],[0,0,0,0],[8.999999E+09,8.999999E+09,8.999999E+09,8.999999E+09,8.999999E+09,8.999999E+09]];
    LOCAL CONST Robtarget Tr_meulage_motif_2_63 := [[96.699390625,82.9637890625,1.6993251953125],[-0.000489514218315733,0.0476030487198184,-0.010271051450657,-0.998813403809994],[0,0,0,0],[8.999999E+09,8.999999E+09,8.999999E+09,8.999999E+09,8.999999E+09,8.999999E+09]];
    LOCAL CONST Robtarget Tr_meulage_motif_2_64 := [[97.405203125,83.6721484375,1.70624011230469],[-0.000489514218315733,0.0476030487198184,-0.010271051450657,-0.998813403809994],[0,0,0,0],[8.999999E+09,8.999999E+09,8.999999E+09,8.999999E+09,8.999999E+09,8.999999E+09]];
    LOCAL CONST Robtarget Tr_meulage_motif_2_65 := [[98.1110234375,84.3805078125,1.71315515136719],[-0.000489514218315733,0.0476030487198184,-0.010271051450657,-0.998813403809994],[0,0,0,0],[8.999999E+09,8.999999E+09,8.999999E+09,8.999999E+09,8.999999E+09,8.999999E+09]];
    LOCAL CONST Robtarget Tr_meulage_motif_2_66 := [[98.8168359375,85.088875,1.72007006835938],[-0.000489514218315733,0.0476030487198184,-0.010271051450657,-0.998813403809994],[0,0,0,0],[8.999999E+09,8.999999E+09,8.999999E+09,8.999999E+09,8.999999E+09,8.999999E+09]];
    LOCAL CONST Robtarget Tr_meulage_motif_2_67 := [[99.5226484375,85.797234375,1.72698498535156],[-0.000489514218315733,0.0476030487198184,-0.010271051450657,-0.998813403809994],[0,0,0,0],[8.999999E+09,8.999999E+09,8.999999E+09,8.999999E+09,8.999999E+09,8.999999E+09]];
    LOCAL CONST Robtarget Tr_meulage_motif_2_68 := [[100.2284609375,86.5056015625,1.73389990234375],[-0.000489514218315733,0.0476030487198184,-0.010271051450657,-0.998813403809994],[0,0,0,0],[8.999999E+09,8.999999E+09,8.999999E+09,8.999999E+09,8.999999E+09,8.999999E+09]];
    LOCAL CONST Robtarget Tr_meulage_motif_2_69 := [[100.93428125,87.2139609375,1.74081494140625],[-0.000489514218315733,0.0476030487198184,-0.010271051450657,-0.998813403809994],[0,0,0,0],[8.999999E+09,8.999999E+09,8.999999E+09,8.999999E+09,8.999999E+09,8.999999E+09]];
    LOCAL CONST Robtarget Tr_meulage_motif_2_70 := [[101.64009375,87.9223203125,1.74772985839844],[-0.000489514218315733,0.0476030487198184,-0.010271051450657,-0.998813403809994],[0,0,0,0],[8.999999E+09,8.999999E+09,8.999999E+09,8.999999E+09,8.999999E+09,8.999999E+09]];
    LOCAL CONST Robtarget Tr_meulage_motif_2_71 := [[102.34590625,88.6306875,1.75464477539063],[-0.000489514218315733,0.0476030487198184,-0.010271051450657,-0.998813403809994],[0,0,0,0],[8.999999E+09,8.999999E+09,8.999999E+09,8.999999E+09,8.999999E+09,8.999999E+09]];
    LOCAL CONST Robtarget Tr_meulage_motif_2_72 := [[103.0517265625,89.339046875,1.76155981445313],[-0.000489514218315733,0.0476030487198184,-0.010271051450657,-0.998813403809994],[0,0,0,0],[8.999999E+09,8.999999E+09,8.999999E+09,8.999999E+09,8.999999E+09,8.999999E+09]];
    LOCAL CONST Robtarget Tr_meulage_motif_2_73 := [[103.7575390625,90.0474140625,1.76847473144531],[-0.000489514218315733,0.0476030487198184,-0.010271051450657,-0.998813403809994],[0,0,0,0],[8.999999E+09,8.999999E+09,8.999999E+09,8.999999E+09,8.999999E+09,8.999999E+09]];
    LOCAL CONST Robtarget Tr_meulage_motif_2_74 := [[104.4633515625,90.7557734375,1.7753896484375],[-0.000489514218315733,0.0476030487198184,-0.010271051450657,-0.998813403809994],[0,0,0,0],[8.999999E+09,8.999999E+09,8.999999E+09,8.999999E+09,8.999999E+09,8.999999E+09]];
    LOCAL CONST Robtarget Tr_meulage_motif_2_75 := [[105.169171875,91.4641328125,1.7823046875],[-0.000489514218315733,0.0476030487198184,-0.010271051450657,-0.998813403809994],[0,0,0,0],[8.999999E+09,8.999999E+09,8.999999E+09,8.999999E+09,8.999999E+09,8.999999E+09]];
    LOCAL CONST Robtarget Tr_meulage_motif_2_76 := [[105.874984375,92.1725,1.78921960449219],[-0.000489514218315733,0.0476030487198184,-0.010271051450657,-0.998813403809994],[0,0,0,0],[8.999999E+09,8.999999E+09,8.999999E+09,8.999999E+09,8.999999E+09,8.999999E+09]];
    LOCAL CONST Robtarget Tr_meulage_motif_2_77 := [[106.580796875,92.880859375,1.79613452148438],[-0.000489514218315733,0.0476030487198184,-0.010271051450657,-0.998813403809994],[0,0,0,0],[8.999999E+09,8.999999E+09,8.999999E+09,8.999999E+09,8.999999E+09,8.999999E+09]];
    LOCAL CONST Robtarget Tr_meulage_motif_2_78 := [[107.2866171875,93.58921875,1.80304943847656],[-0.000489514218315733,0.0476030487198184,-0.010271051450657,-0.998813403809994],[0,0,0,0],[8.999999E+09,8.999999E+09,8.999999E+09,8.999999E+09,8.999999E+09,8.999999E+09]];
    LOCAL CONST Robtarget Tr_meulage_motif_2_79 := [[107.9924296875,94.2975859375,1.80996447753906],[-0.000489514218315733,0.0476030487198184,-0.010271051450657,-0.998813403809994],[0,0,0,0],[8.999999E+09,8.999999E+09,8.999999E+09,8.999999E+09,8.999999E+09,8.999999E+09]];
    LOCAL CONST Robtarget Tr_meulage_motif_2_80 := [[108.6982421875,95.0059453125,1.81687939453125],[-0.000489514218315733,0.0476030487198184,-0.010271051450657,-0.998813403809994],[0,0,0,0],[8.999999E+09,8.999999E+09,8.999999E+09,8.999999E+09,8.999999E+09,8.999999E+09]];
    LOCAL CONST Robtarget Tr_meulage_motif_2_81 := [[109.4040625,95.7143125,1.82379431152344],[-0.000489514218315733,0.0476030487198184,-0.010271051450657,-0.998813403809994],[0,0,0,0],[8.999999E+09,8.999999E+09,8.999999E+09,8.999999E+09,8.999999E+09,8.999999E+09]];
    LOCAL CONST Robtarget Tr_meulage_motif_2_82 := [[110.109875,96.422671875,1.83070935058594],[-0.000489514218315733,0.0476030487198184,-0.010271051450657,-0.998813403809994],[0,0,0,0],[8.999999E+09,8.999999E+09,8.999999E+09,8.999999E+09,8.999999E+09,8.999999E+09]];
    LOCAL CONST Robtarget Tr_meulage_motif_2_83 := [[110.8156875,97.13103125,1.83762426757813],[-0.000489514218315733,0.0476030487198184,-0.010271051450657,-0.998813403809994],[0,0,0,0],[8.999999E+09,8.999999E+09,8.999999E+09,8.999999E+09,8.999999E+09,8.999999E+09]];
    LOCAL CONST Robtarget Tr_meulage_motif_2_84 := [[111.5215078125,97.8393984375,1.84453918457031],[-0.000489514218315733,0.0476030487198184,-0.010271051450657,-0.998813403809994],[0,0,0,0],[8.999999E+09,8.999999E+09,8.999999E+09,8.999999E+09,8.999999E+09,8.999999E+09]];
    LOCAL CONST Robtarget Tr_meulage_motif_2_85 := [[112.2273203125,98.5477578125,1.85145422363281],[-0.000489514218315733,0.0476030487198184,-0.010271051450657,-0.998813403809994],[0,0,0,0],[8.999999E+09,8.999999E+09,8.999999E+09,8.999999E+09,8.999999E+09,8.999999E+09]];
    LOCAL CONST Robtarget Tr_meulage_motif_2_86 := [[112.9331328125,99.256125,1.858369140625],[-0.000489514218315733,0.0476030487198184,-0.010271051450657,-0.998813403809994],[0,0,0,0],[8.999999E+09,8.999999E+09,8.999999E+09,8.999999E+09,8.999999E+09,8.999999E+09]];
    LOCAL CONST Robtarget Tr_meulage_motif_2_87 := [[113.638953125,99.964484375,1.86528405761719],[-0.000489514218315733,0.0476030487198184,-0.010271051450657,-0.998813403809994],[0,0,0,0],[8.999999E+09,8.999999E+09,8.999999E+09,8.999999E+09,8.999999E+09,8.999999E+09]];
    LOCAL CONST Robtarget Tr_meulage_motif_2_88 := [[114.344765625,100.67284375,1.87219897460938],[-0.000489514218315733,0.0476030487198184,-0.010271051450657,-0.998813403809994],[0,0,0,0],[8.999999E+09,8.999999E+09,8.999999E+09,8.999999E+09,8.999999E+09,8.999999E+09]];
    LOCAL CONST Robtarget Tr_meulage_motif_2_89 := [[115.123671875,101.2978828125,1.87827880859375],[-0.000489514218315733,0.0476030487198184,-0.010271051450657,-0.998813403809994],[0,0,0,0],[8.999999E+09,8.999999E+09,8.999999E+09,8.999999E+09,8.999999E+09,8.999999E+09]];
    LOCAL CONST Robtarget Tr_meulage_motif_2_90 := [[115.9413359375,101.819296875,1.88332727050781],[-0.000489514218315733,0.0476030487198184,-0.010271051450657,-0.998813403809994],[0,0,0,0],[8.999999E+09,8.999999E+09,8.999999E+09,8.999999E+09,8.999999E+09,8.999999E+09]];
    LOCAL CONST Robtarget Tr_meulage_motif_2_91 := [[116.735765625,102.23146875,1.88729736328125],[-0.000489514218315733,0.0476030487198184,-0.010271051450657,-0.998813403809994],[0,0,0,0],[8.999999E+09,8.999999E+09,8.999999E+09,8.999999E+09,8.999999E+09,8.999999E+09]];
    LOCAL CONST Robtarget Tr_meulage_motif_2_92 := [[117.4534140625,102.5208046875,1.89006188964844],[-0.000489514218315733,0.0476030487198184,-0.010271051450657,-0.998813403809994],[0,0,0,0],[8.999999E+09,8.999999E+09,8.999999E+09,8.999999E+09,8.999999E+09,8.999999E+09]];
    LOCAL CONST Robtarget Tr_meulage_motif_2_93 := [[118.6528984375,102.785984375,1.89252014160156],[-0.000489514218315733,0.0476030487198184,-0.010271051450657,-0.998813403809994],[0,0,0,0],[8.999999E+09,8.999999E+09,8.999999E+09,8.999999E+09,8.999999E+09,8.999999E+09]];
    LOCAL CONST Robtarget Tr_meulage_motif_2_94 := [[119.9284296875,102.7883125,1.89236547851562],[-0.000489514218315733,0.0476030487198184,-0.010271051450657,-0.998813403809994],[0,0,0,0],[8.999999E+09,8.999999E+09,8.999999E+09,8.999999E+09,8.999999E+09,8.999999E+09]];
    LOCAL CONST Robtarget Tr_meulage_motif_2_95 := [[121.047015625,102.429,1.88865197753906],[-0.000489514218315733,0.0476030487198184,-0.010271051450657,-0.998813403809994],[0,0,0,0],[8.999999E+09,8.999999E+09,8.999999E+09,8.999999E+09,8.999999E+09,8.999999E+09]];
    LOCAL CONST Robtarget Tr_meulage_motif_2_96 := [[121.668515625,102.0706328125,1.88501721191406],[-0.000489514218315733,0.0476030487198184,-0.010271051450657,-0.998813403809994],[0,0,0,0],[8.999999E+09,8.999999E+09,8.999999E+09,8.999999E+09,8.999999E+09,8.999999E+09]];
    LOCAL CONST Robtarget Tr_meulage_motif_2_97 := [[122.2590390625,101.57240625,1.88000207519531],[-0.000489514218315733,0.0476030487198184,-0.010271051450657,-0.998813403809994],[0,0,0,0],[8.999999E+09,8.999999E+09,8.999999E+09,8.999999E+09,8.999999E+09,8.999999E+09]];
    LOCAL CONST Robtarget Tr_meulage_motif_2_98 := [[122.757171875,100.981625,1.87408349609375],[-0.000489514218315733,0.0476030487198184,-0.010271051450657,-0.998813403809994],[0,0,0,0],[8.999999E+09,8.999999E+09,8.999999E+09,8.999999E+09,8.999999E+09,8.999999E+09]];
    LOCAL CONST Robtarget Tr_meulage_motif_2_99 := [[123.24609375,99.90221875,1.86332836914063],[-0.000489514218315733,0.0476030487198184,-0.010271051450657,-0.998813403809994],[0,0,0,0],[8.999999E+09,8.999999E+09,8.999999E+09,8.999999E+09,8.999999E+09,8.999999E+09]];
    LOCAL CONST Robtarget Tr_meulage_motif_2_100 := [[123.3685703125,99.195375,1.85631298828125],[-0.000489514218315733,0.0476030487198184,-0.010271051450657,-0.998813403809994],[0,0,0,0],[8.999999E+09,8.999999E+09,8.999999E+09,8.999999E+09,8.999999E+09,8.999999E+09]];
    LOCAL CONST Robtarget Tr_meulage_motif_2_101 := [[123.370859375,97.9408515625,1.84389196777344],[-0.000489514218315733,0.0476030487198184,-0.010271051450657,-0.998813403809994],[0,0,0,0],[8.999999E+09,8.999999E+09,8.999999E+09,8.999999E+09,8.999999E+09,8.999999E+09]];
    LOCAL CONST Robtarget Tr_meulage_motif_2_102 := [[123.25096875,97.2335625,1.83690588378906],[-0.000489514218315733,0.0476030487198184,-0.010271051450657,-0.998813403809994],[0,0,0,0],[8.999999E+09,8.999999E+09,8.999999E+09,8.999999E+09,8.999999E+09,8.999999E+09]];
    LOCAL CONST Robtarget Tr_meulage_motif_2_103 := [[122.8473671875,96.0576640625,1.82531982421875],[-0.000489514218315733,0.0476030487198184,-0.010271051450657,-0.998813403809994],[0,0,0,0],[8.999999E+09,8.999999E+09,8.999999E+09,8.999999E+09,8.999999E+09,8.999999E+09]];
    LOCAL CONST Robtarget Tr_meulage_motif_2_104 := [[122.473984375,95.2642890625,1.81751684570312],[-0.000489514218315733,0.0476030487198184,-0.010271051450657,-0.998813403809994],[0,0,0,0],[8.999999E+09,8.999999E+09,8.999999E+09,8.999999E+09,8.999999E+09,8.999999E+09]];
    LOCAL CONST Robtarget Tr_meulage_motif_2_105 := [[121.9610078125,94.45978125,1.80962316894531],[-0.000489514218315733,0.0476030487198184,-0.010271051450657,-0.998813403809994],[0,0,0,0],[8.999999E+09,8.999999E+09,8.999999E+09,8.999999E+09,8.999999E+09,8.999999E+09]];
    LOCAL CONST Robtarget Tr_meulage_motif_2_106 := [[121.3451328125,93.6878359375,1.80206616210937],[-0.000489514218315733,0.0476030487198184,-0.010271051450657,-0.998813403809994],[0,0,0,0],[8.999999E+09,8.999999E+09,8.999999E+09,8.999999E+09,8.999999E+09,8.999999E+09]];
    LOCAL CONST Robtarget Tr_meulage_motif_2_107 := [[120.7229140625,92.9066875,1.7944189453125],[-0.000489514218315733,0.0476030487198184,-0.010271051450657,-0.998813403809994],[0,0,0,0],[8.999999E+09,8.999999E+09,8.999999E+09,8.999999E+09,8.999999E+09,8.999999E+09]];
    LOCAL CONST Robtarget Tr_meulage_motif_2_108 := [[120.01709375,92.198328125,1.78750390625],[-0.000489514218315733,0.0476030487198184,-0.010271051450657,-0.998813403809994],[0,0,0,0],[8.999999E+09,8.999999E+09,8.999999E+09,8.999999E+09,8.999999E+09,8.999999E+09]];
    LOCAL CONST Robtarget Tr_meulage_motif_2_109 := [[119.31128125,91.48996875,1.78058898925781],[-0.000489514218315733,0.0476030487198184,-0.010271051450657,-0.998813403809994],[0,0,0,0],[8.999999E+09,8.999999E+09,8.999999E+09,8.999999E+09,8.999999E+09,8.999999E+09]];
    LOCAL CONST Robtarget Tr_meulage_motif_2_110 := [[118.60546875,90.7816015625,1.77367407226563],[-0.000489514218315733,0.0476030487198184,-0.010271051450657,-0.998813403809994],[0,0,0,0],[8.999999E+09,8.999999E+09,8.999999E+09,8.999999E+09,8.999999E+09,8.999999E+09]];
    LOCAL CONST Robtarget Tr_meulage_motif_2_111 := [[117.8996484375,90.0732421875,1.76675915527344],[-0.000489514218315733,0.0476030487198184,-0.010271051450657,-0.998813403809994],[0,0,0,0],[8.999999E+09,8.999999E+09,8.999999E+09,8.999999E+09,8.999999E+09,8.999999E+09]];
    LOCAL CONST Robtarget Tr_meulage_motif_2_112 := [[117.1938359375,89.364875,1.75984411621094],[-0.000489514218315733,0.0476030487198184,-0.010271051450657,-0.998813403809994],[0,0,0,0],[8.999999E+09,8.999999E+09,8.999999E+09,8.999999E+09,8.999999E+09,8.999999E+09]];
    LOCAL CONST Robtarget Tr_meulage_motif_2_113 := [[116.4880234375,88.656515625,1.75292919921875],[-0.000489514218315733,0.0476030487198184,-0.010271051450657,-0.998813403809994],[0,0,0,0],[8.999999E+09,8.999999E+09,8.999999E+09,8.999999E+09,8.999999E+09,8.999999E+09]];
    LOCAL CONST Robtarget Tr_meulage_motif_2_114 := [[115.782203125,87.94815625,1.74601428222656],[-0.000489514218315733,0.0476030487198184,-0.010271051450657,-0.998813403809994],[0,0,0,0],[8.999999E+09,8.999999E+09,8.999999E+09,8.999999E+09,8.999999E+09,8.999999E+09]];
    LOCAL CONST Robtarget Tr_meulage_motif_2_115 := [[115.076390625,87.2397890625,1.73909924316406],[-0.000489514218315733,0.0476030487198184,-0.010271051450657,-0.998813403809994],[0,0,0,0],[8.999999E+09,8.999999E+09,8.999999E+09,8.999999E+09,8.999999E+09,8.999999E+09]];
    LOCAL CONST Robtarget Tr_meulage_motif_2_116 := [[114.370578125,86.5314296875,1.73218432617188],[-0.000489514218315733,0.0476030487198184,-0.010271051450657,-0.998813403809994],[0,0,0,0],[8.999999E+09,8.999999E+09,8.999999E+09,8.999999E+09,8.999999E+09,8.999999E+09]];
    LOCAL CONST Robtarget Tr_meulage_motif_2_117 := [[113.664765625,85.8230625,1.72526940917969],[-0.000489514218315733,0.0476030487198184,-0.010271051450657,-0.998813403809994],[0,0,0,0],[8.999999E+09,8.999999E+09,8.999999E+09,8.999999E+09,8.999999E+09,8.999999E+09]];
    LOCAL CONST Robtarget Tr_meulage_motif_2_118 := [[112.9589453125,85.114703125,1.71835437011719],[-0.000489514218315733,0.0476030487198184,-0.010271051450657,-0.998813403809994],[0,0,0,0],[8.999999E+09,8.999999E+09,8.999999E+09,8.999999E+09,8.999999E+09,8.999999E+09]];
    LOCAL CONST Robtarget Tr_meulage_motif_2_119 := [[112.2531328125,84.40634375,1.711439453125],[-0.000489514218315733,0.0476030487198184,-0.010271051450657,-0.998813403809994],[0,0,0,0],[8.999999E+09,8.999999E+09,8.999999E+09,8.999999E+09,8.999999E+09,8.999999E+09]];
    LOCAL CONST Robtarget Tr_meulage_motif_2_120 := [[111.5473203125,83.6979765625,1.70452453613281],[-0.000489514218315733,0.0476030487198184,-0.010271051450657,-0.998813403809994],[0,0,0,0],[8.999999E+09,8.999999E+09,8.999999E+09,8.999999E+09,8.999999E+09,8.999999E+09]];
    LOCAL CONST Robtarget Tr_meulage_motif_2_121 := [[110.8415,82.9896171875,1.69760961914063],[-0.000489514218315733,0.0476030487198184,-0.010271051450657,-0.998813403809994],[0,0,0,0],[8.999999E+09,8.999999E+09,8.999999E+09,8.999999E+09,8.999999E+09,8.999999E+09]];
    LOCAL CONST Robtarget Tr_meulage_motif_2_122 := [[110.1356875,82.28125,1.69069458007813],[-0.000489514218315733,0.0476030487198184,-0.010271051450657,-0.998813403809994],[0,0,0,0],[8.999999E+09,8.999999E+09,8.999999E+09,8.999999E+09,8.999999E+09,8.999999E+09]];
    LOCAL CONST Robtarget Tr_meulage_motif_2_123 := [[109.429875,81.572890625,1.68377966308594],[-0.000489514218315733,0.0476030487198184,-0.010271051450657,-0.998813403809994],[0,0,0,0],[8.999999E+09,8.999999E+09,8.999999E+09,8.999999E+09,8.999999E+09,8.999999E+09]];
    LOCAL CONST Robtarget Tr_meulage_motif_2_124 := [[108.7240546875,80.86453125,1.67686474609375],[-0.000489514218315733,0.0476030487198184,-0.010271051450657,-0.998813403809994],[0,0,0,0],[8.999999E+09,8.999999E+09,8.999999E+09,8.999999E+09,8.999999E+09,8.999999E+09]];
    LOCAL CONST Robtarget Tr_meulage_motif_2_125 := [[108.0182421875,80.1561640625,1.66994970703125],[-0.000489514218315733,0.0476030487198184,-0.010271051450657,-0.998813403809994],[0,0,0,0],[8.999999E+09,8.999999E+09,8.999999E+09,8.999999E+09,8.999999E+09,8.999999E+09]];
    LOCAL CONST Robtarget Tr_meulage_motif_2_126 := [[107.3124296875,79.4478046875,1.66303479003906],[-0.000489514218315733,0.0476030487198184,-0.010271051450657,-0.998813403809994],[0,0,0,0],[8.999999E+09,8.999999E+09,8.999999E+09,8.999999E+09,8.999999E+09,8.999999E+09]];
    LOCAL CONST Robtarget Tr_meulage_motif_2_127 := [[106.606609375,78.7394375,1.65611987304688],[-0.000489514218315733,0.0476030487198184,-0.010271051450657,-0.998813403809994],[0,0,0,0],[8.999999E+09,8.999999E+09,8.999999E+09,8.999999E+09,8.999999E+09,8.999999E+09]];
    LOCAL CONST Robtarget Tr_meulage_motif_2_128 := [[105.900796875,78.031078125,1.64920495605469],[-0.000489514218315733,0.0476030487198184,-0.010271051450657,-0.998813403809994],[0,0,0,0],[8.999999E+09,8.999999E+09,8.999999E+09,8.999999E+09,8.999999E+09,8.999999E+09]];
    LOCAL CONST Robtarget Tr_meulage_motif_2_129 := [[105.194984375,77.32271875,1.64228991699219],[-0.000489514218315733,0.0476030487198184,-0.010271051450657,-0.998813403809994],[0,0,0,0],[8.999999E+09,8.999999E+09,8.999999E+09,8.999999E+09,8.999999E+09,8.999999E+09]];
    LOCAL CONST Robtarget Tr_meulage_motif_2_130 := [[104.4891640625,76.6143515625,1.635375],[-0.000489514218315733,0.0476030487198184,-0.010271051450657,-0.998813403809994],[0,0,0,0],[8.999999E+09,8.999999E+09,8.999999E+09,8.999999E+09,8.999999E+09,8.999999E+09]];
    LOCAL CONST Robtarget Tr_meulage_motif_2_131 := [[103.7833515625,75.9059921875,1.62846008300781],[-0.000489514218315733,0.0476030487198184,-0.010271051450657,-0.998813403809994],[0,0,0,0],[8.999999E+09,8.999999E+09,8.999999E+09,8.999999E+09,8.999999E+09,8.999999E+09]];
    LOCAL CONST Robtarget Tr_meulage_motif_2_132 := [[103.0775390625,75.197625,1.62154504394531],[-0.000489514218315733,0.0476030487198184,-0.010271051450657,-0.998813403809994],[0,0,0,0],[8.999999E+09,8.999999E+09,8.999999E+09,8.999999E+09,8.999999E+09,8.999999E+09]];
    LOCAL CONST Robtarget Tr_meulage_motif_2_133 := [[102.37171875,74.489265625,1.61463012695313],[-0.000489514218315733,0.0476030487198184,-0.010271051450657,-0.998813403809994],[0,0,0,0],[8.999999E+09,8.999999E+09,8.999999E+09,8.999999E+09,8.999999E+09,8.999999E+09]];
    LOCAL CONST Robtarget Tr_meulage_motif_2_134 := [[101.66590625,73.78090625,1.60771520996094],[-0.000489514218315733,0.0476030487198184,-0.010271051450657,-0.998813403809994],[0,0,0,0],[8.999999E+09,8.999999E+09,8.999999E+09,8.999999E+09,8.999999E+09,8.999999E+09]];
    LOCAL CONST Robtarget Tr_meulage_motif_2_135 := [[100.96009375,73.0725390625,1.60080017089844],[-0.000489514218315733,0.0476030487198184,-0.010271051450657,-0.998813403809994],[0,0,0,0],[8.999999E+09,8.999999E+09,8.999999E+09,8.999999E+09,8.999999E+09,8.999999E+09]];
    LOCAL CONST Robtarget Tr_meulage_motif_2_136 := [[100.2542734375,72.3641796875,1.59388525390625],[-0.000489514218315733,0.0476030487198184,-0.010271051450657,-0.998813403809994],[0,0,0,0],[8.999999E+09,8.999999E+09,8.999999E+09,8.999999E+09,8.999999E+09,8.999999E+09]];
    LOCAL CONST Robtarget Tr_meulage_motif_2_137 := [[99.5484609375,71.6558125,1.58697033691406],[-0.000489514218315733,0.0476030487198184,-0.010271051450657,-0.998813403809994],[0,0,0,0],[8.999999E+09,8.999999E+09,8.999999E+09,8.999999E+09,8.999999E+09,8.999999E+09]];
    LOCAL CONST Robtarget Tr_meulage_motif_2_138 := [[98.9262421875,70.8746640625,1.57932312011719],[-0.000489514218315733,0.0476030487198184,-0.010271051450657,-0.998813403809994],[0,0,0,0],[8.999999E+09,8.999999E+09,8.999999E+09,8.999999E+09,8.999999E+09,8.999999E+09]];
    LOCAL CONST Robtarget Tr_meulage_motif_2_139 := [[98.4077890625,70.0551484375,1.57128149414063],[-0.000489514218315733,0.0476030487198184,-0.010271051450657,-0.998813403809994],[0,0,0,0],[8.999999E+09,8.999999E+09,8.999999E+09,8.999999E+09,8.999999E+09,8.999999E+09]];
    LOCAL CONST Robtarget Tr_meulage_motif_2_140 := [[97.9985,69.2592578125,1.56345849609375],[-0.000489514218315733,0.0476030487198184,-0.010271051450657,-0.998813403809994],[0,0,0,0],[8.999999E+09,8.999999E+09,8.999999E+09,8.999999E+09,8.999999E+09,8.999999E+09]];
    LOCAL CONST Robtarget Tr_meulage_motif_2_141 := [[97.66465625,68.5332734375,1.5563173828125],[-0.000489514218315733,0.0476030487198184,-0.010271051450657,-0.998813403809994],[0,0,0,0],[8.999999E+09,8.999999E+09,8.999999E+09,8.999999E+09,8.999999E+09,8.999999E+09]];
    LOCAL CONST Robtarget Tr_meulage_motif_2_142 := [[97.3239765625,67.3184765625,1.54433740234375],[-0.000489514218315733,0.0476030487198184,-0.010271051450657,-0.998813403809994],[0,0,0,0],[8.999999E+09,8.999999E+09,8.999999E+09,8.999999E+09,8.999999E+09,8.999999E+09]];
    LOCAL CONST Robtarget Tr_meulage_motif_2_143 := [[97.20178125,65.9949453125,1.53125036621094],[-0.000489514218315733,0.0476030487198184,-0.010271051450657,-0.998813403809994],[0,0,0,0],[8.999999E+09,8.999999E+09,8.999999E+09,8.999999E+09,8.999999E+09,8.999999E+09]];
    LOCAL CONST Robtarget Tr_meulage_motif_2_144 := [[97.3288046875,64.6718671875,1.51813317871094],[-0.000489514218315733,0.0476030487198184,-0.010271051450657,-0.998813403809994],[0,0,0,0],[8.999999E+09,8.999999E+09,8.999999E+09,8.999999E+09,8.999999E+09,8.999999E+09]];
    LOCAL CONST Robtarget Tr_meulage_motif_2_145 := [[97.7749609375,63.53829296875,1.50684765625],[-0.000489514218315733,0.0476030487198184,-0.010271051450657,-0.998813403809994],[0,0,0,0],[8.999999E+09,8.999999E+09,8.999999E+09,8.999999E+09,8.999999E+09,8.999999E+09]];
    LOCAL CONST Robtarget Tr_meulage_motif_2_146 := [[98.2488828125,63.027921875,1.50172863769531],[-0.000489514218315733,0.0476030487198184,-0.010271051450657,-0.998813403809994],[0,0,0,0],[8.999999E+09,8.999999E+09,8.999999E+09,8.999999E+09,8.999999E+09,8.999999E+09]];
    LOCAL CONST Robtarget Tr_meulage_motif_2_147 := [[98.7173046875,62.5612265625,1.49704260253906],[-0.000489514218315733,0.0476030487198184,-0.010271051450657,-0.998813403809994],[0,0,0,0],[8.999999E+09,8.999999E+09,8.999999E+09,8.999999E+09,8.999999E+09,8.999999E+09]];
    LOCAL CONST Robtarget Tr_meulage_motif_2_148 := [[99.2243515625,62.13351171875,1.49273718261719],[-0.000489514218315733,0.0476030487198184,-0.010271051450657,-0.998813403809994],[0,0,0,0],[8.999999E+09,8.999999E+09,8.999999E+09,8.999999E+09,8.999999E+09,8.999999E+09]];
    LOCAL CONST Robtarget Tr_meulage_motif_2_149 := [[100.3564765625,61.7088359375,1.48837487792969],[-0.000489514218315733,0.0476030487198184,-0.010271051450657,-0.998813403809994],[0,0,0,0],[8.999999E+09,8.999999E+09,8.999999E+09,8.999999E+09,8.999999E+09,8.999999E+09]];
    LOCAL CONST Robtarget Tr_meulage_motif_2_150 := [[101.6741875,61.60518359375,1.48716491699219],[-0.000489514218315733,0.0476030487198184,-0.010271051450657,-0.998813403809994],[0,0,0,0],[8.999999E+09,8.999999E+09,8.999999E+09,8.999999E+09,8.999999E+09,8.999999E+09]];
    LOCAL CONST Robtarget Tr_meulage_motif_2_151 := [[102.9836953125,61.74512109375,1.48836779785156],[-0.000489514218315733,0.0476030487198184,-0.010271051450657,-0.998813403809994],[0,0,0,0],[8.999999E+09,8.999999E+09,8.999999E+09,8.999999E+09,8.999999E+09,8.999999E+09]];
    LOCAL CONST Robtarget Tr_meulage_motif_2_152 := [[103.7490078125,61.9525234375,1.49031457519531],[-0.000489514218315733,0.0476030487198184,-0.010271051450657,-0.998813403809994],[0,0,0,0],[8.999999E+09,8.999999E+09,8.999999E+09,8.999999E+09,8.999999E+09,8.999999E+09]];
    LOCAL CONST Robtarget Tr_meulage_motif_2_153 := [[104.9118125,62.428828125,1.49486828613281],[-0.000489514218315733,0.0476030487198184,-0.010271051450657,-0.998813403809994],[0,0,0,0],[8.999999E+09,8.999999E+09,8.999999E+09,8.999999E+09,8.999999E+09,8.999999E+09]];
    LOCAL CONST Robtarget Tr_meulage_motif_2_154 := [[105.6953359375,62.8410234375,1.49884008789062],[-0.000489514218315733,0.0476030487198184,-0.010271051450657,-0.998813403809994],[0,0,0,0],[8.999999E+09,8.999999E+09,8.999999E+09,8.999999E+09,8.999999E+09,8.999999E+09]];
    LOCAL CONST Robtarget Tr_meulage_motif_2_155 := [[106.498,63.35690625,1.5038359375],[-0.000489514218315733,0.0476030487198184,-0.010271051450657,-0.998813403809994],[0,0,0,0],[8.999999E+09,8.999999E+09,8.999999E+09,8.999999E+09,8.999999E+09,8.999999E+09]];
    LOCAL CONST Robtarget Tr_meulage_motif_2_156 := [[107.2677265625,63.97556640625,1.50985375976562],[-0.000489514218315733,0.0476030487198184,-0.010271051450657,-0.998813403809994],[0,0,0,0],[8.999999E+09,8.999999E+09,8.999999E+09,8.999999E+09,8.999999E+09,8.999999E+09]];
    LOCAL CONST Robtarget Tr_meulage_motif_2_157 := [[108.0466328125,64.60060546875,1.51593359375],[-0.000489514218315733,0.0476030487198184,-0.010271051450657,-0.998813403809994],[0,0,0,0],[8.999999E+09,8.999999E+09,8.999999E+09,8.999999E+09,8.999999E+09,8.999999E+09]];
    LOCAL CONST Robtarget Tr_meulage_motif_2_158 := [[108.752453125,65.30896875,1.52284851074219],[-0.000489514218315733,0.0476030487198184,-0.010271051450657,-0.998813403809994],[0,0,0,0],[8.999999E+09,8.999999E+09,8.999999E+09,8.999999E+09,8.999999E+09,8.999999E+09]];
    LOCAL CONST Robtarget Tr_meulage_motif_2_159 := [[109.458265625,66.017328125,1.52976354980469],[-0.000489514218315733,0.0476030487198184,-0.010271051450657,-0.998813403809994],[0,0,0,0],[8.999999E+09,8.999999E+09,8.999999E+09,8.999999E+09,8.999999E+09,8.999999E+09]];
    LOCAL CONST Robtarget Tr_meulage_motif_2_160 := [[110.164078125,66.7256953125,1.53667846679688],[-0.000489514218315733,0.0476030487198184,-0.010271051450657,-0.998813403809994],[0,0,0,0],[8.999999E+09,8.999999E+09,8.999999E+09,8.999999E+09,8.999999E+09,8.999999E+09]];
    LOCAL CONST Robtarget Tr_meulage_motif_2_161 := [[110.8698984375,67.4340546875,1.54359338378906],[-0.000489514218315733,0.0476030487198184,-0.010271051450657,-0.998813403809994],[0,0,0,0],[8.999999E+09,8.999999E+09,8.999999E+09,8.999999E+09,8.999999E+09,8.999999E+09]];
    LOCAL CONST Robtarget Tr_meulage_motif_2_162 := [[111.5757109375,68.1424140625,1.55050830078125],[-0.000489514218315733,0.0476030487198184,-0.010271051450657,-0.998813403809994],[0,0,0,0],[8.999999E+09,8.999999E+09,8.999999E+09,8.999999E+09,8.999999E+09,8.999999E+09]];
    LOCAL CONST Robtarget Tr_meulage_motif_2_163 := [[112.2815234375,68.85078125,1.55742333984375],[-0.000489514218315733,0.0476030487198184,-0.010271051450657,-0.998813403809994],[0,0,0,0],[8.999999E+09,8.999999E+09,8.999999E+09,8.999999E+09,8.999999E+09,8.999999E+09]];
    LOCAL CONST Robtarget Tr_meulage_motif_2_164 := [[112.98734375,69.559140625,1.56433825683594],[-0.000489514218315733,0.0476030487198184,-0.010271051450657,-0.998813403809994],[0,0,0,0],[8.999999E+09,8.999999E+09,8.999999E+09,8.999999E+09,8.999999E+09,8.999999E+09]];
    LOCAL CONST Robtarget Tr_meulage_motif_2_165 := [[113.69315625,70.2675078125,1.57125317382813],[-0.000489514218315733,0.0476030487198184,-0.010271051450657,-0.998813403809994],[0,0,0,0],[8.999999E+09,8.999999E+09,8.999999E+09,8.999999E+09,8.999999E+09,8.999999E+09]];
    LOCAL CONST Robtarget Tr_meulage_motif_2_166 := [[114.39896875,70.9758671875,1.57816821289062],[-0.000489514218315733,0.0476030487198184,-0.010271051450657,-0.998813403809994],[0,0,0,0],[8.999999E+09,8.999999E+09,8.999999E+09,8.999999E+09,8.999999E+09,8.999999E+09]];
    LOCAL CONST Robtarget Tr_meulage_motif_2_167 := [[115.1047890625,71.6842265625,1.58508312988281],[-0.000489514218315733,0.0476030487198184,-0.010271051450657,-0.998813403809994],[0,0,0,0],[8.999999E+09,8.999999E+09,8.999999E+09,8.999999E+09,8.999999E+09,8.999999E+09]];
    LOCAL CONST Robtarget Tr_meulage_motif_2_168 := [[115.8106015625,72.39259375,1.591998046875],[-0.000489514218315733,0.0476030487198184,-0.010271051450657,-0.998813403809994],[0,0,0,0],[8.999999E+09,8.999999E+09,8.999999E+09,8.999999E+09,8.999999E+09,8.999999E+09]];
    LOCAL CONST Robtarget Tr_meulage_motif_2_169 := [[116.5164140625,73.100953125,1.5989130859375],[-0.000489514218315733,0.0476030487198184,-0.010271051450657,-0.998813403809994],[0,0,0,0],[8.999999E+09,8.999999E+09,8.999999E+09,8.999999E+09,8.999999E+09,8.999999E+09]];
    LOCAL CONST Robtarget Tr_meulage_motif_2_170 := [[117.2222265625,73.8093203125,1.60582800292969],[-0.000489514218315733,0.0476030487198184,-0.010271051450657,-0.998813403809994],[0,0,0,0],[8.999999E+09,8.999999E+09,8.999999E+09,8.999999E+09,8.999999E+09,8.999999E+09]];
    LOCAL CONST Robtarget Tr_meulage_motif_2_171 := [[117.928046875,74.5176796875,1.61274291992188],[-0.000489514218315733,0.0476030487198184,-0.010271051450657,-0.998813403809994],[0,0,0,0],[8.999999E+09,8.999999E+09,8.999999E+09,8.999999E+09,8.999999E+09,8.999999E+09]];
    LOCAL CONST Robtarget Tr_meulage_motif_2_172 := [[118.633859375,75.2260390625,1.61965783691406],[-0.000489514218315733,0.0476030487198184,-0.010271051450657,-0.998813403809994],[0,0,0,0],[8.999999E+09,8.999999E+09,8.999999E+09,8.999999E+09,8.999999E+09,8.999999E+09]];
    LOCAL CONST Robtarget Tr_meulage_motif_2_173 := [[119.339671875,75.93440625,1.62657287597656],[-0.000489514218315733,0.0476030487198184,-0.010271051450657,-0.998813403809994],[0,0,0,0],[8.999999E+09,8.999999E+09,8.999999E+09,8.999999E+09,8.999999E+09,8.999999E+09]];
    LOCAL CONST Robtarget Tr_meulage_motif_2_174 := [[120.0454921875,76.642765625,1.63348779296875],[-0.000489514218315733,0.0476030487198184,-0.010271051450657,-0.998813403809994],[0,0,0,0],[8.999999E+09,8.999999E+09,8.999999E+09,8.999999E+09,8.999999E+09,8.999999E+09]];
    LOCAL CONST Robtarget Tr_meulage_motif_2_175 := [[120.7513046875,77.3511328125,1.64040270996094],[-0.000489514218315733,0.0476030487198184,-0.010271051450657,-0.998813403809994],[0,0,0,0],[8.999999E+09,8.999999E+09,8.999999E+09,8.999999E+09,8.999999E+09,8.999999E+09]];
    LOCAL CONST Robtarget Tr_meulage_motif_2_176 := [[121.4571171875,78.0594921875,1.64731774902344],[-0.000489514218315733,0.0476030487198184,-0.010271051450657,-0.998813403809994],[0,0,0,0],[8.999999E+09,8.999999E+09,8.999999E+09,8.999999E+09,8.999999E+09,8.999999E+09]];
    LOCAL CONST Robtarget Tr_meulage_motif_2_177 := [[122.1629375,78.7678515625,1.65423266601563],[-0.000489514218315733,0.0476030487198184,-0.010271051450657,-0.998813403809994],[0,0,0,0],[8.999999E+09,8.999999E+09,8.999999E+09,8.999999E+09,8.999999E+09,8.999999E+09]];
    LOCAL CONST Robtarget Tr_meulage_motif_2_178 := [[122.86875,79.47621875,1.66114758300781],[-0.000489514218315733,0.0476030487198184,-0.010271051450657,-0.998813403809994],[0,0,0,0],[8.999999E+09,8.999999E+09,8.999999E+09,8.999999E+09,8.999999E+09,8.999999E+09]];
    LOCAL CONST Robtarget Tr_meulage_motif_2_179 := [[123.5745625,80.184578125,1.6680625],[-0.000489514218315733,0.0476030487198184,-0.010271051450657,-0.998813403809994],[0,0,0,0],[8.999999E+09,8.999999E+09,8.999999E+09,8.999999E+09,8.999999E+09,8.999999E+09]];
    LOCAL CONST Robtarget Tr_meulage_motif_2_180 := [[124.2803828125,80.8929453125,1.6749775390625],[-0.000489514218315733,0.0476030487198184,-0.010271051450657,-0.998813403809994],[0,0,0,0],[8.999999E+09,8.999999E+09,8.999999E+09,8.999999E+09,8.999999E+09,8.999999E+09]];
    LOCAL CONST Robtarget Tr_meulage_motif_2_181 := [[124.9861953125,81.6013046875,1.68189245605469],[-0.000489514218315733,0.0476030487198184,-0.010271051450657,-0.998813403809994],[0,0,0,0],[8.999999E+09,8.999999E+09,8.999999E+09,8.999999E+09,8.999999E+09,8.999999E+09]];
    LOCAL CONST Robtarget Tr_meulage_motif_2_182 := [[125.6920078125,82.3096640625,1.68880737304688],[-0.000489514218315733,0.0476030487198184,-0.010271051450657,-0.998813403809994],[0,0,0,0],[8.999999E+09,8.999999E+09,8.999999E+09,8.999999E+09,8.999999E+09,8.999999E+09]];
    LOCAL CONST Robtarget Tr_meulage_motif_2_183 := [[126.397828125,83.01803125,1.69572241210938],[-0.000489514218315733,0.0476030487198184,-0.010271051450657,-0.998813403809994],[0,0,0,0],[8.999999E+09,8.999999E+09,8.999999E+09,8.999999E+09,8.999999E+09,8.999999E+09]];
    LOCAL CONST Robtarget Tr_meulage_motif_2_184 := [[127.103640625,83.726390625,1.70263732910156],[-0.000489514218315733,0.0476030487198184,-0.010271051450657,-0.998813403809994],[0,0,0,0],[8.999999E+09,8.999999E+09,8.999999E+09,8.999999E+09,8.999999E+09,8.999999E+09]];
    LOCAL CONST Robtarget Tr_meulage_motif_2_185 := [[127.809453125,84.4347578125,1.70955224609375],[-0.000489514218315733,0.0476030487198184,-0.010271051450657,-0.998813403809994],[0,0,0,0],[8.999999E+09,8.999999E+09,8.999999E+09,8.999999E+09,8.999999E+09,8.999999E+09]];
    LOCAL CONST Robtarget Tr_meulage_motif_2_186 := [[128.5152734375,85.1431171875,1.71646728515625],[-0.000489514218315733,0.0476030487198184,-0.010271051450657,-0.998813403809994],[0,0,0,0],[8.999999E+09,8.999999E+09,8.999999E+09,8.999999E+09,8.999999E+09,8.999999E+09]];
    LOCAL CONST Robtarget Tr_meulage_motif_2_187 := [[129.2210859375,85.8514765625,1.72338220214844],[-0.000489514218315733,0.0476030487198184,-0.010271051450657,-0.998813403809994],[0,0,0,0],[8.999999E+09,8.999999E+09,8.999999E+09,8.999999E+09,8.999999E+09,8.999999E+09]];
    LOCAL CONST Robtarget Tr_meulage_motif_2_188 := [[129.9999921875,86.476515625,1.72946203613281],[-0.000489514218315733,0.0476030487198184,-0.010271051450657,-0.998813403809994],[0,0,0,0],[8.999999E+09,8.999999E+09,8.999999E+09,8.999999E+09,8.999999E+09,8.999999E+09]];
    LOCAL CONST Robtarget Tr_meulage_motif_2_189 := [[130.81765625,86.9979296875,1.73451037597656],[-0.000489514218315733,0.0476030487198184,-0.010271051450657,-0.998813403809994],[0,0,0,0],[8.999999E+09,8.999999E+09,8.999999E+09,8.999999E+09,8.999999E+09,8.999999E+09]];
    LOCAL CONST Robtarget Tr_meulage_motif_2_190 := [[131.61209375,87.4101015625,1.73848046875],[-0.000489514218315733,0.0476030487198184,-0.010271051450657,-0.998813403809994],[0,0,0,0],[8.999999E+09,8.999999E+09,8.999999E+09,8.999999E+09,8.999999E+09,8.999999E+09]];
    LOCAL CONST Robtarget Tr_meulage_motif_2_191 := [[132.329734375,87.6994453125,1.74124523925781],[-0.000489514218315733,0.0476030487198184,-0.010271051450657,-0.998813403809994],[0,0,0,0],[8.999999E+09,8.999999E+09,8.999999E+09,8.999999E+09,8.999999E+09,8.999999E+09]];
    LOCAL CONST Robtarget Tr_meulage_motif_2_192 := [[133.529203125,87.964625,1.74370349121094],[-0.000489514218315733,0.0476030487198184,-0.010271051450657,-0.998813403809994],[0,0,0,0],[8.999999E+09,8.999999E+09,8.999999E+09,8.999999E+09,8.999999E+09,8.999999E+09]];
    LOCAL CONST Robtarget Tr_meulage_motif_2_193 := [[134.80475,87.9669453125,1.74354858398437],[-0.000489514218315733,0.0476030487198184,-0.010271051450657,-0.998813403809994],[0,0,0,0],[8.999999E+09,8.999999E+09,8.999999E+09,8.999999E+09,8.999999E+09,8.999999E+09]];
    LOCAL CONST Robtarget Tr_meulage_motif_2_194 := [[135.923328125,87.607640625,1.73983532714844],[-0.000489514218315733,0.0476030487198184,-0.010271051450657,-0.998813403809994],[0,0,0,0],[8.999999E+09,8.999999E+09,8.999999E+09,8.999999E+09,8.999999E+09,8.999999E+09]];
    LOCAL CONST Robtarget Tr_meulage_motif_2_195 := [[136.544828125,87.249265625,1.73620043945312],[-0.000489514218315733,0.0476030487198184,-0.010271051450657,-0.998813403809994],[0,0,0,0],[8.999999E+09,8.999999E+09,8.999999E+09,8.999999E+09,8.999999E+09,8.999999E+09]];
    LOCAL CONST Robtarget Tr_meulage_motif_2_196 := [[137.135359375,86.7510390625,1.73118530273438],[-0.000489514218315733,0.0476030487198184,-0.010271051450657,-0.998813403809994],[0,0,0,0],[8.999999E+09,8.999999E+09,8.999999E+09,8.999999E+09,8.999999E+09,8.999999E+09]];
    LOCAL CONST Robtarget Tr_meulage_motif_2_197 := [[137.633484375,86.160265625,1.72526672363281],[-0.000489514218315733,0.0476030487198184,-0.010271051450657,-0.998813403809994],[0,0,0,0],[8.999999E+09,8.999999E+09,8.999999E+09,8.999999E+09,8.999999E+09,8.999999E+09]];
    LOCAL CONST Robtarget Tr_meulage_motif_2_198 := [[138.12240625,85.0808671875,1.71451171875],[-0.000489514218315733,0.0476030487198184,-0.010271051450657,-0.998813403809994],[0,0,0,0],[8.999999E+09,8.999999E+09,8.999999E+09,8.999999E+09,8.999999E+09,8.999999E+09]];
    LOCAL CONST Robtarget Tr_meulage_motif_2_199 := [[138.244875,84.374015625,1.70749621582031],[-0.000489514218315733,0.0476030487198184,-0.010271051450657,-0.998813403809994],[0,0,0,0],[8.999999E+09,8.999999E+09,8.999999E+09,8.999999E+09,8.999999E+09,8.999999E+09]];
    LOCAL CONST Robtarget Tr_meulage_motif_2_200 := [[138.2471875,83.11946875,1.69507495117188],[-0.000489514218315733,0.0476030487198184,-0.010271051450657,-0.998813403809994],[0,0,0,0],[8.999999E+09,8.999999E+09,8.999999E+09,8.999999E+09,8.999999E+09,8.999999E+09]];
    LOCAL CONST Robtarget Tr_meulage_motif_2_201 := [[138.12728125,82.412203125,1.68808911132813],[-0.000489514218315733,0.0476030487198184,-0.010271051450657,-0.998813403809994],[0,0,0,0],[8.999999E+09,8.999999E+09,8.999999E+09,8.999999E+09,8.999999E+09,8.999999E+09]];
    LOCAL CONST Robtarget Tr_meulage_motif_2_202 := [[137.723703125,81.2362890625,1.6765029296875],[-0.000489514218315733,0.0476030487198184,-0.010271051450657,-0.998813403809994],[0,0,0,0],[8.999999E+09,8.999999E+09,8.999999E+09,8.999999E+09,8.999999E+09,8.999999E+09]];
    LOCAL CONST Robtarget Tr_meulage_motif_2_203 := [[137.3503125,80.44290625,1.66869995117187],[-0.000489514218315733,0.0476030487198184,-0.010271051450657,-0.998813403809994],[0,0,0,0],[8.999999E+09,8.999999E+09,8.999999E+09,8.999999E+09,8.999999E+09,8.999999E+09]];
    LOCAL CONST Robtarget Tr_meulage_motif_2_204 := [[136.83734375,79.6383984375,1.66080615234375],[-0.000489514218315733,0.0476030487198184,-0.010271051450657,-0.998813403809994],[0,0,0,0],[8.999999E+09,8.999999E+09,8.999999E+09,8.999999E+09,8.999999E+09,8.999999E+09]];
    LOCAL CONST Robtarget Tr_meulage_motif_2_205 := [[136.2214375,78.866484375,1.65324938964844],[-0.000489514218315733,0.0476030487198184,-0.010271051450657,-0.998813403809994],[0,0,0,0],[8.999999E+09,8.999999E+09,8.999999E+09,8.999999E+09,8.999999E+09,8.999999E+09]];
    LOCAL CONST Robtarget Tr_meulage_motif_2_206 := [[135.599234375,78.0853203125,1.64560205078125],[-0.000489514218315733,0.0476030487198184,-0.010271051450657,-0.998813403809994],[0,0,0,0],[8.999999E+09,8.999999E+09,8.999999E+09,8.999999E+09,8.999999E+09,8.999999E+09]];
    LOCAL CONST Robtarget Tr_meulage_motif_2_207 := [[134.893421875,77.3769609375,1.63868713378906],[-0.000489514218315733,0.0476030487198184,-0.010271051450657,-0.998813403809994],[0,0,0,0],[8.999999E+09,8.999999E+09,8.999999E+09,8.999999E+09,8.999999E+09,8.999999E+09]];
    LOCAL CONST Robtarget Tr_meulage_motif_2_208 := [[134.187609375,76.6686015625,1.63177221679688],[-0.000489514218315733,0.0476030487198184,-0.010271051450657,-0.998813403809994],[0,0,0,0],[8.999999E+09,8.999999E+09,8.999999E+09,8.999999E+09,8.999999E+09,8.999999E+09]];
    LOCAL CONST Robtarget Tr_meulage_motif_2_209 := [[133.48178125,75.960234375,1.62485717773437],[-0.000489514218315733,0.0476030487198184,-0.010271051450657,-0.998813403809994],[0,0,0,0],[8.999999E+09,8.999999E+09,8.999999E+09,8.999999E+09,8.999999E+09,8.999999E+09]];
    LOCAL CONST Robtarget Tr_meulage_motif_2_210 := [[132.77596875,75.251875,1.61794226074219],[-0.000489514218315733,0.0476030487198184,-0.010271051450657,-0.998813403809994],[0,0,0,0],[8.999999E+09,8.999999E+09,8.999999E+09,8.999999E+09,8.999999E+09,8.999999E+09]];
    LOCAL CONST Robtarget Tr_meulage_motif_2_211 := [[132.07015625,74.5435078125,1.61102734375],[-0.000489514218315733,0.0476030487198184,-0.010271051450657,-0.998813403809994],[0,0,0,0],[8.999999E+09,8.999999E+09,8.999999E+09,8.999999E+09,8.999999E+09,8.999999E+09]];
    LOCAL CONST Robtarget Tr_meulage_motif_2_212 := [[131.36434375,73.8351484375,1.6041123046875],[-0.000489514218315733,0.0476030487198184,-0.010271051450657,-0.998813403809994],[0,0,0,0],[8.999999E+09,8.999999E+09,8.999999E+09,8.999999E+09,8.999999E+09,8.999999E+09]];
    LOCAL CONST Robtarget Tr_meulage_motif_2_213 := [[130.6585234375,73.1267890625,1.59719738769531],[-0.000489514218315733,0.0476030487198184,-0.010271051450657,-0.998813403809994],[0,0,0,0],[8.999999E+09,8.999999E+09,8.999999E+09,8.999999E+09,8.999999E+09,8.999999E+09]];
    LOCAL CONST Robtarget Tr_meulage_motif_2_214 := [[129.9527109375,72.418421875,1.59028247070313],[-0.000489514218315733,0.0476030487198184,-0.010271051450657,-0.998813403809994],[0,0,0,0],[8.999999E+09,8.999999E+09,8.999999E+09,8.999999E+09,8.999999E+09,8.999999E+09]];
    LOCAL CONST Robtarget Tr_meulage_motif_2_215 := [[129.2468984375,71.7100625,1.58336743164062],[-0.000489514218315733,0.0476030487198184,-0.010271051450657,-0.998813403809994],[0,0,0,0],[8.999999E+09,8.999999E+09,8.999999E+09,8.999999E+09,8.999999E+09,8.999999E+09]];
    LOCAL CONST Robtarget Tr_meulage_motif_2_216 := [[128.5410859375,71.0016953125,1.57645251464844],[-0.000489514218315733,0.0476030487198184,-0.010271051450657,-0.998813403809994],[0,0,0,0],[8.999999E+09,8.999999E+09,8.999999E+09,8.999999E+09,8.999999E+09,8.999999E+09]];
    LOCAL CONST Robtarget Tr_meulage_motif_2_217 := [[127.835265625,70.2933359375,1.56953759765625],[-0.000489514218315733,0.0476030487198184,-0.010271051450657,-0.998813403809994],[0,0,0,0],[8.999999E+09,8.999999E+09,8.999999E+09,8.999999E+09,8.999999E+09,8.999999E+09]];
    LOCAL CONST Robtarget Tr_meulage_motif_2_218 := [[127.129453125,69.5849765625,1.56262268066406],[-0.000489514218315733,0.0476030487198184,-0.010271051450657,-0.998813403809994],[0,0,0,0],[8.999999E+09,8.999999E+09,8.999999E+09,8.999999E+09,8.999999E+09,8.999999E+09]];
    LOCAL CONST Robtarget Tr_meulage_motif_2_219 := [[126.423640625,68.876609375,1.55570764160156],[-0.000489514218315733,0.0476030487198184,-0.010271051450657,-0.998813403809994],[0,0,0,0],[8.999999E+09,8.999999E+09,8.999999E+09,8.999999E+09,8.999999E+09,8.999999E+09]];
    LOCAL CONST Robtarget Tr_meulage_motif_2_220 := [[125.7178203125,68.16825,1.54879272460938],[-0.000489514218315733,0.0476030487198184,-0.010271051450657,-0.998813403809994],[0,0,0,0],[8.999999E+09,8.999999E+09,8.999999E+09,8.999999E+09,8.999999E+09,8.999999E+09]];
    LOCAL CONST Robtarget Tr_meulage_motif_2_221 := [[125.0120078125,67.4598828125,1.54187780761719],[-0.000489514218315733,0.0476030487198184,-0.010271051450657,-0.998813403809994],[0,0,0,0],[8.999999E+09,8.999999E+09,8.999999E+09,8.999999E+09,8.999999E+09,8.999999E+09]];
    LOCAL CONST Robtarget Tr_meulage_motif_2_222 := [[124.3061953125,66.7515234375,1.53496276855469],[-0.000489514218315733,0.0476030487198184,-0.010271051450657,-0.998813403809994],[0,0,0,0],[8.999999E+09,8.999999E+09,8.999999E+09,8.999999E+09,8.999999E+09,8.999999E+09]];
    LOCAL CONST Robtarget Tr_meulage_motif_2_223 := [[123.600375,66.0431640625,1.5280478515625],[-0.000489514218315733,0.0476030487198184,-0.010271051450657,-0.998813403809994],[0,0,0,0],[8.999999E+09,8.999999E+09,8.999999E+09,8.999999E+09,8.999999E+09,8.999999E+09]];
    LOCAL CONST Robtarget Tr_meulage_motif_2_224 := [[122.8945625,65.334796875,1.52113293457031],[-0.000489514218315733,0.0476030487198184,-0.010271051450657,-0.998813403809994],[0,0,0,0],[8.999999E+09,8.999999E+09,8.999999E+09,8.999999E+09,8.999999E+09,8.999999E+09]];
    LOCAL CONST Robtarget Tr_meulage_motif_2_225 := [[122.18875,64.6264375,1.51421801757813],[-0.000489514218315733,0.0476030487198184,-0.010271051450657,-0.998813403809994],[0,0,0,0],[8.999999E+09,8.999999E+09,8.999999E+09,8.999999E+09,8.999999E+09,8.999999E+09]];
    LOCAL CONST Robtarget Tr_meulage_motif_2_226 := [[121.4829296875,63.91807421875,1.50730297851563],[-0.000489514218315733,0.0476030487198184,-0.010271051450657,-0.998813403809994],[0,0,0,0],[8.999999E+09,8.999999E+09,8.999999E+09,8.999999E+09,8.999999E+09,8.999999E+09]];
    LOCAL CONST Robtarget Tr_meulage_motif_2_227 := [[120.7771171875,63.2097109375,1.50038806152344],[-0.000489514218315733,0.0476030487198184,-0.010271051450657,-0.998813403809994],[0,0,0,0],[8.999999E+09,8.999999E+09,8.999999E+09,8.999999E+09,8.999999E+09,8.999999E+09]];
    LOCAL CONST Robtarget Tr_meulage_motif_2_228 := [[120.0713046875,62.50134765625,1.49347314453125],[-0.000489514218315733,0.0476030487198184,-0.010271051450657,-0.998813403809994],[0,0,0,0],[8.999999E+09,8.999999E+09,8.999999E+09,8.999999E+09,8.999999E+09,8.999999E+09]];
    LOCAL CONST Robtarget Tr_meulage_motif_2_229 := [[119.365484375,61.792984375,1.48655810546875],[-0.000489514218315733,0.0476030487198184,-0.010271051450657,-0.998813403809994],[0,0,0,0],[8.999999E+09,8.999999E+09,8.999999E+09,8.999999E+09,8.999999E+09,8.999999E+09]];
    LOCAL CONST Robtarget Tr_meulage_motif_2_230 := [[118.659671875,61.084625,1.47964318847656],[-0.000489514218315733,0.0476030487198184,-0.010271051450657,-0.998813403809994],[0,0,0,0],[8.999999E+09,8.999999E+09,8.999999E+09,8.999999E+09,8.999999E+09,8.999999E+09]];
    LOCAL CONST Robtarget Tr_meulage_motif_2_231 := [[117.953859375,60.37626171875,1.47272827148438],[-0.000489514218315733,0.0476030487198184,-0.010271051450657,-0.998813403809994],[0,0,0,0],[8.999999E+09,8.999999E+09,8.999999E+09,8.999999E+09,8.999999E+09,8.999999E+09]];
    LOCAL CONST Robtarget Tr_meulage_motif_2_232 := [[117.2480390625,59.6678984375,1.46581323242188],[-0.000489514218315733,0.0476030487198184,-0.010271051450657,-0.998813403809994],[0,0,0,0],[8.999999E+09,8.999999E+09,8.999999E+09,8.999999E+09,8.999999E+09,8.999999E+09]];
    LOCAL CONST Robtarget Tr_meulage_motif_2_233 := [[116.5422265625,58.95953515625,1.45889831542969],[-0.000489514218315733,0.0476030487198184,-0.010271051450657,-0.998813403809994],[0,0,0,0],[8.999999E+09,8.999999E+09,8.999999E+09,8.999999E+09,8.999999E+09,8.999999E+09]];
    LOCAL CONST Robtarget Tr_meulage_motif_2_234 := [[115.8364140625,58.251171875,1.4519833984375],[-0.000489514218315733,0.0476030487198184,-0.010271051450657,-0.998813403809994],[0,0,0,0],[8.999999E+09,8.999999E+09,8.999999E+09,8.999999E+09,8.999999E+09,8.999999E+09]];
    LOCAL CONST Robtarget Tr_meulage_motif_2_235 := [[115.1306015625,57.5428125,1.44506848144531],[-0.000489514218315733,0.0476030487198184,-0.010271051450657,-0.998813403809994],[0,0,0,0],[8.999999E+09,8.999999E+09,8.999999E+09,8.999999E+09,8.999999E+09,8.999999E+09]];
    LOCAL CONST Robtarget Tr_meulage_motif_2_236 := [[114.42478125,56.83444921875,1.43815344238281],[-0.000489514218315733,0.0476030487198184,-0.010271051450657,-0.998813403809994],[0,0,0,0],[8.999999E+09,8.999999E+09,8.999999E+09,8.999999E+09,8.999999E+09,8.999999E+09]];
    LOCAL CONST Robtarget Tr_meulage_motif_2_237 := [[113.8025703125,56.0532890625,1.43050610351563],[-0.000489514218315733,0.0476030487198184,-0.010271051450657,-0.998813403809994],[0,0,0,0],[8.999999E+09,8.999999E+09,8.999999E+09,8.999999E+09,8.999999E+09,8.999999E+09]];
    LOCAL CONST Robtarget Tr_meulage_motif_2_238 := [[113.284125,55.2337734375,1.42246447753906],[-0.000489514218315733,0.0476030487198184,-0.010271051450657,-0.998813403809994],[0,0,0,0],[8.999999E+09,8.999999E+09,8.999999E+09,8.999999E+09,8.999999E+09,8.999999E+09]];
    LOCAL CONST Robtarget Tr_meulage_motif_2_239 := [[112.8748203125,54.43788671875,1.41464172363281],[-0.000489514218315733,0.0476030487198184,-0.010271051450657,-0.998813403809994],[0,0,0,0],[8.999999E+09,8.999999E+09,8.999999E+09,8.999999E+09,8.999999E+09,8.999999E+09]];
    LOCAL CONST Robtarget Tr_meulage_motif_2_240 := [[112.5880859375,53.71923046875,1.40756640625],[-0.000489514218315733,0.0476030487198184,-0.010271051450657,-0.998813403809994],[0,0,0,0],[8.999999E+09,8.999999E+09,8.999999E+09,8.999999E+09,8.999999E+09,8.999999E+09]];
    LOCAL CONST Robtarget Tr_meulage_motif_2_241 := [[112.32728125,52.5188515625,1.39571813964844],[-0.000489514218315733,0.0476030487198184,-0.010271051450657,-0.998813403809994],[0,0,0,0],[8.999999E+09,8.999999E+09,8.999999E+09,8.999999E+09,8.999999E+09,8.999999E+09]];
    LOCAL CONST Robtarget Tr_meulage_motif_2_242 := [[112.41928125,51.27976171875,1.38343725585938],[-0.000489514218315733,0.0476030487198184,-0.010271051450657,-0.998813403809994],[0,0,0,0],[8.999999E+09,8.999999E+09,8.999999E+09,8.999999E+09,8.999999E+09,8.999999E+09]];
    LOCAL CONST Robtarget Tr_meulage_motif_2_243 := [[112.8763359375,50.3268984375,1.373939453125],[-0.000489514218315733,0.0476030487198184,-0.010271051450657,-0.998813403809994],[0,0,0,0],[8.999999E+09,8.999999E+09,8.999999E+09,8.999999E+09,8.999999E+09,8.999999E+09]];
    LOCAL CONST Robtarget Tr_meulage_motif_2_244 := [[113.292234375,49.95440234375,1.37019348144531],[-0.000489514218315733,0.0476030487198184,-0.010271051450657,-0.998813403809994],[0,0,0,0],[8.999999E+09,8.999999E+09,8.999999E+09,8.999999E+09,8.999999E+09,8.999999E+09]];
    LOCAL CONST Robtarget Tr_meulage_motif_2_245 := [[113.585234375,49.6563984375,1.3672021484375],[-0.000489514218315733,0.0476030487198184,-0.010271051450657,-0.998813403809994],[0,0,0,0],[8.999999E+09,8.999999E+09,8.999999E+09,8.999999E+09,8.999999E+09,8.999999E+09]];
    LOCAL CONST Robtarget Tr_meulage_motif_2_246 := [[114.527515625,49.2288046875,1.36283728027344],[-0.000489514218315733,0.0476030487198184,-0.010271051450657,-0.998813403809994],[0,0,0,0],[8.999999E+09,8.999999E+09,8.999999E+09,8.999999E+09,8.999999E+09,8.999999E+09]];
    LOCAL CONST Robtarget Tr_meulage_motif_2_247 := [[115.7577421875,49.16334765625,1.36201782226562],[-0.000489514218315733,0.0476030487198184,-0.010271051450657,-0.998813403809994],[0,0,0,0],[8.999999E+09,8.999999E+09,8.999999E+09,8.999999E+09,8.999999E+09,8.999999E+09]];
    LOCAL CONST Robtarget Tr_meulage_motif_2_248 := [[116.4893828125,49.2985078125,1.36325402832031],[-0.000489514218315733,0.0476030487198184,-0.010271051450657,-0.998813403809994],[0,0,0,0],[8.999999E+09,8.999999E+09,8.999999E+09,8.999999E+09,8.999999E+09,8.999999E+09]];
    LOCAL CONST Robtarget Tr_meulage_motif_2_249 := [[117.6629453125,49.724796875,1.36731103515625],[-0.000489514218315733,0.0476030487198184,-0.010271051450657,-0.998813403809994],[0,0,0,0],[8.999999E+09,8.999999E+09,8.999999E+09,8.999999E+09,8.999999E+09,8.999999E+09]];
    LOCAL CONST Robtarget Tr_meulage_motif_2_250 := [[118.4464765625,50.136984375,1.37128271484375],[-0.000489514218315733,0.0476030487198184,-0.010271051450657,-0.998813403809994],[0,0,0,0],[8.999999E+09,8.999999E+09,8.999999E+09,8.999999E+09,8.999999E+09,8.999999E+09]];
    LOCAL CONST Robtarget Tr_meulage_motif_2_251 := [[119.2491484375,50.65285546875,1.3762783203125],[-0.000489514218315733,0.0476030487198184,-0.010271051450657,-0.998813403809994],[0,0,0,0],[8.999999E+09,8.999999E+09,8.999999E+09,8.999999E+09,8.999999E+09,8.999999E+09]];
    LOCAL CONST Robtarget Tr_meulage_motif_2_252 := [[120.01884375,51.271546875,1.38229663085937],[-0.000489514218315733,0.0476030487198184,-0.010271051450657,-0.998813403809994],[0,0,0,0],[8.999999E+09,8.999999E+09,8.999999E+09,8.999999E+09,8.999999E+09,8.999999E+09]];
    LOCAL CONST Robtarget Tr_meulage_motif_2_253 := [[120.797765625,51.89657421875,1.38837634277344],[-0.000489514218315733,0.0476030487198184,-0.010271051450657,-0.998813403809994],[0,0,0,0],[8.999999E+09,8.999999E+09,8.999999E+09,8.999999E+09,8.999999E+09,8.999999E+09]];
    LOCAL CONST Robtarget Tr_meulage_motif_2_254 := [[121.5035859375,52.6049375,1.39529125976563],[-0.000489514218315733,0.0476030487198184,-0.010271051450657,-0.998813403809994],[0,0,0,0],[8.999999E+09,8.999999E+09,8.999999E+09,8.999999E+09,8.999999E+09,8.999999E+09]];
    LOCAL CONST Robtarget Tr_meulage_motif_2_255 := [[122.2093984375,53.31330078125,1.40220617675781],[-0.000489514218315733,0.0476030487198184,-0.010271051450657,-0.998813403809994],[0,0,0,0],[8.999999E+09,8.999999E+09,8.999999E+09,8.999999E+09,8.999999E+09,8.999999E+09]];
    LOCAL CONST Robtarget Tr_meulage_motif_2_256 := [[122.9152109375,54.0216640625,1.40912121582031],[-0.000489514218315733,0.0476030487198184,-0.010271051450657,-0.998813403809994],[0,0,0,0],[8.999999E+09,8.999999E+09,8.999999E+09,8.999999E+09,8.999999E+09,8.999999E+09]];
    LOCAL CONST Robtarget Tr_meulage_motif_2_257 := [[123.62103125,54.73002734375,1.4160361328125],[-0.000489514218315733,0.0476030487198184,-0.010271051450657,-0.998813403809994],[0,0,0,0],[8.999999E+09,8.999999E+09,8.999999E+09,8.999999E+09,8.999999E+09,8.999999E+09]];
    LOCAL CONST Robtarget Tr_meulage_motif_2_258 := [[124.32684375,55.43838671875,1.42295104980469],[-0.000489514218315733,0.0476030487198184,-0.010271051450657,-0.998813403809994],[0,0,0,0],[8.999999E+09,8.999999E+09,8.999999E+09,8.999999E+09,8.999999E+09,8.999999E+09]];
    LOCAL CONST Robtarget Tr_meulage_motif_2_259 := [[125.03265625,56.14675,1.42986596679687],[-0.000489514218315733,0.0476030487198184,-0.010271051450657,-0.998813403809994],[0,0,0,0],[8.999999E+09,8.999999E+09,8.999999E+09,8.999999E+09,8.999999E+09,8.999999E+09]];
    LOCAL CONST Robtarget Tr_meulage_motif_2_260 := [[125.73846875,56.85511328125,1.43678100585938],[-0.000489514218315733,0.0476030487198184,-0.010271051450657,-0.998813403809994],[0,0,0,0],[8.999999E+09,8.999999E+09,8.999999E+09,8.999999E+09,8.999999E+09,8.999999E+09]];
    LOCAL CONST Robtarget Tr_meulage_motif_2_261 := [[126.4442890625,57.5634765625,1.44369592285156],[-0.000489514218315733,0.0476030487198184,-0.010271051450657,-0.998813403809994],[0,0,0,0],[8.999999E+09,8.999999E+09,8.999999E+09,8.999999E+09,8.999999E+09,8.999999E+09]];
    LOCAL CONST Robtarget Tr_meulage_motif_2_262 := [[127.1501015625,58.27183984375,1.45061083984375],[-0.000489514218315733,0.0476030487198184,-0.010271051450657,-0.998813403809994],[0,0,0,0],[8.999999E+09,8.999999E+09,8.999999E+09,8.999999E+09,8.999999E+09,8.999999E+09]];
    LOCAL CONST Robtarget Tr_meulage_motif_2_263 := [[127.8559140625,58.98019921875,1.45752587890625],[-0.000489514218315733,0.0476030487198184,-0.010271051450657,-0.998813403809994],[0,0,0,0],[8.999999E+09,8.999999E+09,8.999999E+09,8.999999E+09,8.999999E+09,8.999999E+09]];
    LOCAL CONST Robtarget Tr_meulage_motif_2_264 := [[128.561734375,59.6885625,1.46444079589844],[-0.000489514218315733,0.0476030487198184,-0.010271051450657,-0.998813403809994],[0,0,0,0],[8.999999E+09,8.999999E+09,8.999999E+09,8.999999E+09,8.999999E+09,8.999999E+09]];
    LOCAL CONST Robtarget Tr_meulage_motif_2_265 := [[129.267546875,60.39692578125,1.47135571289062],[-0.000489514218315733,0.0476030487198184,-0.010271051450657,-0.998813403809994],[0,0,0,0],[8.999999E+09,8.999999E+09,8.999999E+09,8.999999E+09,8.999999E+09,8.999999E+09]];
    LOCAL CONST Robtarget Tr_meulage_motif_2_266 := [[129.973359375,61.1052890625,1.47827075195313],[-0.000489514218315733,0.0476030487198184,-0.010271051450657,-0.998813403809994],[0,0,0,0],[8.999999E+09,8.999999E+09,8.999999E+09,8.999999E+09,8.999999E+09,8.999999E+09]];
    LOCAL CONST Robtarget Tr_meulage_motif_2_267 := [[130.6791796875,61.81365234375,1.48518566894531],[-0.000489514218315733,0.0476030487198184,-0.010271051450657,-0.998813403809994],[0,0,0,0],[8.999999E+09,8.999999E+09,8.999999E+09,8.999999E+09,8.999999E+09,8.999999E+09]];
    LOCAL CONST Robtarget Tr_meulage_motif_2_268 := [[131.384984375,62.52201171875,1.4921005859375],[-0.000489514218315733,0.0476030487198184,-0.010271051450657,-0.998813403809994],[0,0,0,0],[8.999999E+09,8.999999E+09,8.999999E+09,8.999999E+09,8.999999E+09,8.999999E+09]];
    LOCAL CONST Robtarget Tr_meulage_motif_2_269 := [[132.0908125,63.230375,1.49901550292969],[-0.000489514218315733,0.0476030487198184,-0.010271051450657,-0.998813403809994],[0,0,0,0],[8.999999E+09,8.999999E+09,8.999999E+09,8.999999E+09,8.999999E+09,8.999999E+09]];
    LOCAL CONST Robtarget Tr_meulage_motif_2_270 := [[132.796625,63.93873828125,1.50593054199219],[-0.000489514218315733,0.0476030487198184,-0.010271051450657,-0.998813403809994],[0,0,0,0],[8.999999E+09,8.999999E+09,8.999999E+09,8.999999E+09,8.999999E+09,8.999999E+09]];
    LOCAL CONST Robtarget Tr_meulage_motif_2_271 := [[133.5024375,64.6471015625,1.51284545898437],[-0.000489514218315733,0.0476030487198184,-0.010271051450657,-0.998813403809994],[0,0,0,0],[8.999999E+09,8.999999E+09,8.999999E+09,8.999999E+09,8.999999E+09,8.999999E+09]];
    LOCAL CONST Robtarget Tr_meulage_motif_2_272 := [[134.20825,65.35546484375,1.51976037597656],[-0.000489514218315733,0.0476030487198184,-0.010271051450657,-0.998813403809994],[0,0,0,0],[8.999999E+09,8.999999E+09,8.999999E+09,8.999999E+09,8.999999E+09,8.999999E+09]];
    LOCAL CONST Robtarget Tr_meulage_motif_2_273 := [[134.9140625,66.063828125,1.52667541503906],[-0.000489514218315733,0.0476030487198184,-0.010271051450657,-0.998813403809994],[0,0,0,0],[8.999999E+09,8.999999E+09,8.999999E+09,8.999999E+09,8.999999E+09,8.999999E+09]];
    LOCAL CONST Robtarget Tr_meulage_motif_2_274 := [[135.619875,66.7721875,1.53359033203125],[-0.000489514218315733,0.0476030487198184,-0.010271051450657,-0.998813403809994],[0,0,0,0],[8.999999E+09,8.999999E+09,8.999999E+09,8.999999E+09,8.999999E+09,8.999999E+09]];
    LOCAL CONST Robtarget Tr_meulage_motif_2_275 := [[136.325703125,67.480546875,1.54050524902344],[-0.000489514218315733,0.0476030487198184,-0.010271051450657,-0.998813403809994],[0,0,0,0],[8.999999E+09,8.999999E+09,8.999999E+09,8.999999E+09,8.999999E+09,8.999999E+09]];
    LOCAL CONST Robtarget Tr_meulage_motif_2_276 := [[137.031515625,68.1889140625,1.54742016601563],[-0.000489514218315733,0.0476030487198184,-0.010271051450657,-0.998813403809994],[0,0,0,0],[8.999999E+09,8.999999E+09,8.999999E+09,8.999999E+09,8.999999E+09,8.999999E+09]];
    LOCAL CONST Robtarget Tr_meulage_motif_2_277 := [[137.737328125,68.8972734375,1.55433520507812],[-0.000489514218315733,0.0476030487198184,-0.010271051450657,-0.998813403809994],[0,0,0,0],[8.999999E+09,8.999999E+09,8.999999E+09,8.999999E+09,8.999999E+09,8.999999E+09]];
    LOCAL CONST Robtarget Tr_meulage_motif_2_278 := [[138.443140625,69.605640625,1.56125012207031],[-0.000489514218315733,0.0476030487198184,-0.010271051450657,-0.998813403809994],[0,0,0,0],[8.999999E+09,8.999999E+09,8.999999E+09,8.999999E+09,8.999999E+09,8.999999E+09]];
    LOCAL CONST Robtarget Tr_meulage_motif_2_279 := [[139.148953125,70.314,1.5681650390625],[-0.000489514218315733,0.0476030487198184,-0.010271051450657,-0.998813403809994],[0,0,0,0],[8.999999E+09,8.999999E+09,8.999999E+09,8.999999E+09,8.999999E+09,8.999999E+09]];
    LOCAL CONST Robtarget Tr_meulage_motif_2_280 := [[139.854765625,71.022359375,1.575080078125],[-0.000489514218315733,0.0476030487198184,-0.010271051450657,-0.998813403809994],[0,0,0,0],[8.999999E+09,8.999999E+09,8.999999E+09,8.999999E+09,8.999999E+09,8.999999E+09]];
    LOCAL CONST Robtarget Tr_meulage_motif_2_281 := [[140.56059375,71.7307265625,1.58199499511719],[-0.000489514218315733,0.0476030487198184,-0.010271051450657,-0.998813403809994],[0,0,0,0],[8.999999E+09,8.999999E+09,8.999999E+09,8.999999E+09,8.999999E+09,8.999999E+09]];
    LOCAL CONST Robtarget Tr_meulage_motif_2_282 := [[141.26640625,72.4390859375,1.58890991210938],[-0.000489514218315733,0.0476030487198184,-0.010271051450657,-0.998813403809994],[0,0,0,0],[8.999999E+09,8.999999E+09,8.999999E+09,8.999999E+09,8.999999E+09,8.999999E+09]];
    LOCAL CONST Robtarget Tr_meulage_motif_2_283 := [[141.97221875,73.147453125,1.59582495117187],[-0.000489514218315733,0.0476030487198184,-0.010271051450657,-0.998813403809994],[0,0,0,0],[8.999999E+09,8.999999E+09,8.999999E+09,8.999999E+09,8.999999E+09,8.999999E+09]];
    LOCAL CONST Robtarget Tr_meulage_motif_2_284 := [[142.67803125,73.8558125,1.60273986816406],[-0.000489514218315733,0.0476030487198184,-0.010271051450657,-0.998813403809994],[0,0,0,0],[8.999999E+09,8.999999E+09,8.999999E+09,8.999999E+09,8.999999E+09,8.999999E+09]];
    LOCAL CONST Robtarget Tr_meulage_motif_2_285 := [[143.38384375,74.564171875,1.60965478515625],[-0.000489514218315733,0.0476030487198184,-0.010271051450657,-0.998813403809994],[0,0,0,0],[8.999999E+09,8.999999E+09,8.999999E+09,8.999999E+09,8.999999E+09,8.999999E+09]];
    LOCAL CONST Robtarget Tr_meulage_motif_2_286 := [[144.08965625,75.2725390625,1.61656970214844],[-0.000489514218315733,0.0476030487198184,-0.010271051450657,-0.998813403809994],[0,0,0,0],[8.999999E+09,8.999999E+09,8.999999E+09,8.999999E+09,8.999999E+09,8.999999E+09]];
    LOCAL CONST Robtarget Tr_meulage_motif_2_287 := [[144.795484375,75.9808984375,1.62348474121094],[-0.000489514218315733,0.0476030487198184,-0.010271051450657,-0.998813403809994],[0,0,0,0],[8.999999E+09,8.999999E+09,8.999999E+09,8.999999E+09,8.999999E+09,8.999999E+09]];
    LOCAL CONST Robtarget Tr_meulage_motif_2_288 := [[145.501296875,76.689265625,1.63039965820313],[-0.000489514218315733,0.0476030487198184,-0.010271051450657,-0.998813403809994],[0,0,0,0],[8.999999E+09,8.999999E+09,8.999999E+09,8.999999E+09,8.999999E+09,8.999999E+09]];
    LOCAL CONST Robtarget Tr_meulage_motif_2_289 := [[146.207109375,77.397625,1.63731457519531],[-0.000489514218315733,0.0476030487198184,-0.010271051450657,-0.998813403809994],[0,0,0,0],[8.999999E+09,8.999999E+09,8.999999E+09,8.999999E+09,8.999999E+09,8.999999E+09]];
    LOCAL CONST Robtarget Tr_meulage_motif_2_290 := [[146.912921875,78.105984375,1.64422961425781],[-0.000489514218315733,0.0476030487198184,-0.010271051450657,-0.998813403809994],[0,0,0,0],[8.999999E+09,8.999999E+09,8.999999E+09,8.999999E+09,8.999999E+09,8.999999E+09]];
    LOCAL CONST Robtarget Tr_meulage_motif_2_291 := [[147.618734375,78.8143515625,1.65114453125],[-0.000489514218315733,0.0476030487198184,-0.010271051450657,-0.998813403809994],[0,0,0,0],[8.999999E+09,8.999999E+09,8.999999E+09,8.999999E+09,8.999999E+09,8.999999E+09]];
    LOCAL CONST Robtarget Tr_meulage_motif_2_292 := [[148.324546875,79.5227109375,1.65805944824219],[-0.000489514218315733,0.0476030487198184,-0.010271051450657,-0.998813403809994],[0,0,0,0],[8.999999E+09,8.999999E+09,8.999999E+09,8.999999E+09,8.999999E+09,8.999999E+09]];
    LOCAL CONST Robtarget Tr_meulage_motif_2_293 := [[149.030359375,80.231078125,1.66497436523438],[-0.000489514218315733,0.0476030487198184,-0.010271051450657,-0.998813403809994],[0,0,0,0],[8.999999E+09,8.999999E+09,8.999999E+09,8.999999E+09,8.999999E+09,8.999999E+09]];
